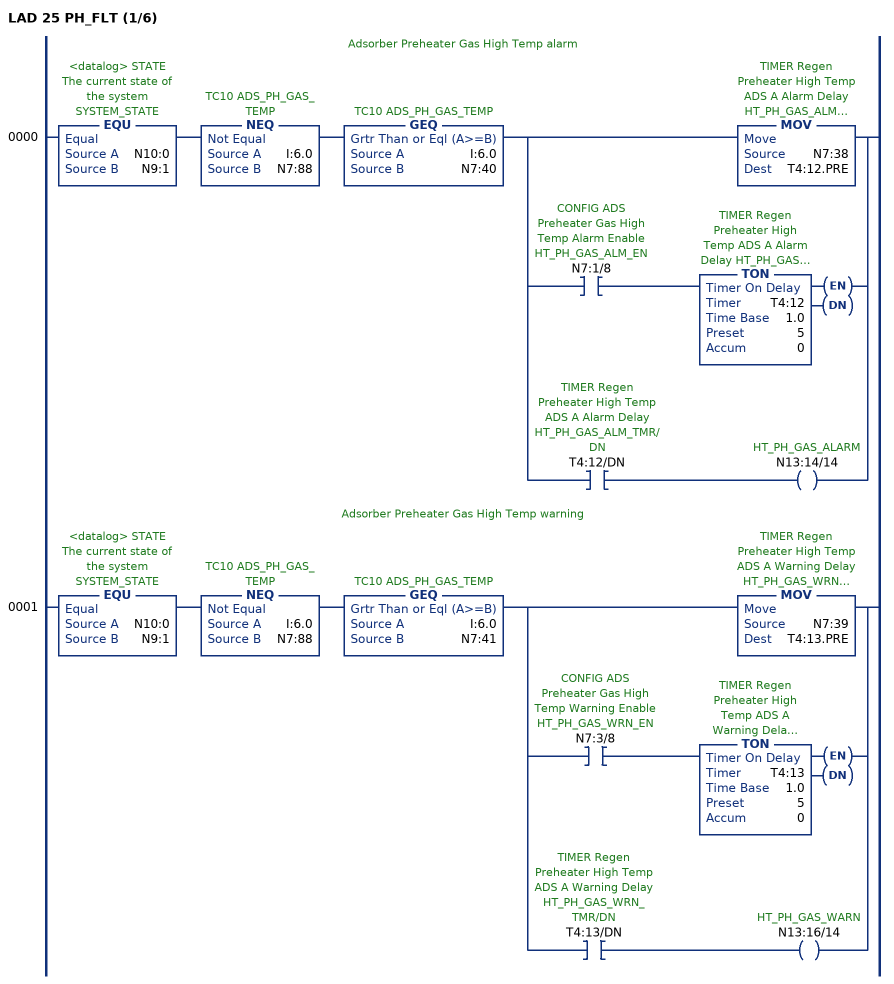
% Rung: 0 %
% Adsorber Preheater Gas High Temp alarm %
SOR EQU N10:0 N9:1 NEQ I:6.0 N7:88 GEQ I:6.0 N7:40 BST MOV N7:38 T4:12.PRE NXB XIC N7:1/8 TON T4:12 1.0 5 0 NXB XIC T4:12/DN OTE N13:14/14 BND EOR
%   N10:0  SYSTEM_STATE  "<datalog> STATE The current state of the system" %
%   N9:1  SYSTEM_PROCESS  "STATE System Process" %
%   I:6.0  ADS_PH_GAS_TEMP  "TC10" %
%   N7:88  TC_OPEN_SP  "CONFIG TC Open Setpoint" %
%   N7:40  HT_PH_GAS_ALM_SP  "CONFIG ADS Preheater Gas High Temp Alarm Setpoint" %
%   N7:38  HT_PH_GAS_ALM_DLY  "CONFIG ADS Preheater Gas High Temp Alarm Delay" %
%   T4:12  HT_PH_GAS_ALM_TMR  "TIMER Regen Preheater High Temp ADS A Alarm Delay" %
%   N7:1/8  HT_PH_GAS_ALM_EN  "CONFIG ADS Preheater Gas High Temp Alarm Enable" %
%   N13:14/14  HT_PH_GAS_ALARM %
% Rung: 1 %
% Adsorber Preheater Gas High Temp warning %
SOR EQU N10:0 N9:1 NEQ I:6.0 N7:88 GEQ I:6.0 N7:41 BST MOV N7:39 T4:13.PRE NXB XIC N7:3/8 TON T4:13 1.0 5 0 NXB XIC T4:13/DN OTE N13:16/14 BND EOR
%   N10:0  SYSTEM_STATE  "<datalog> STATE The current state of the system" %
%   N9:1  SYSTEM_PROCESS  "STATE System Process" %
%   I:6.0  ADS_PH_GAS_TEMP  "TC10" %
%   N7:88  TC_OPEN_SP  "CONFIG TC Open Setpoint" %
%   N7:41  HT_PH_GAS_WRN_SP  "CONFIG ADS Preheater Gas High Temp Warning Setpoint" %
%   N7:39  HT_PH_GAS_WRN_DLY  "CONFIG ADS Preheater Gas High Temp Warning Delay" %
%   T4:13  HT_PH_GAS_WRN_TMR  "TIMER Regen Preheater High Temp ADS A Warning Delay" %
%   N7:3/8  HT_PH_GAS_WRN_EN  "CONFIG ADS Preheater Gas High Temp Warning Enable" %
%   N13:16/14  HT_PH_GAS_WARN %

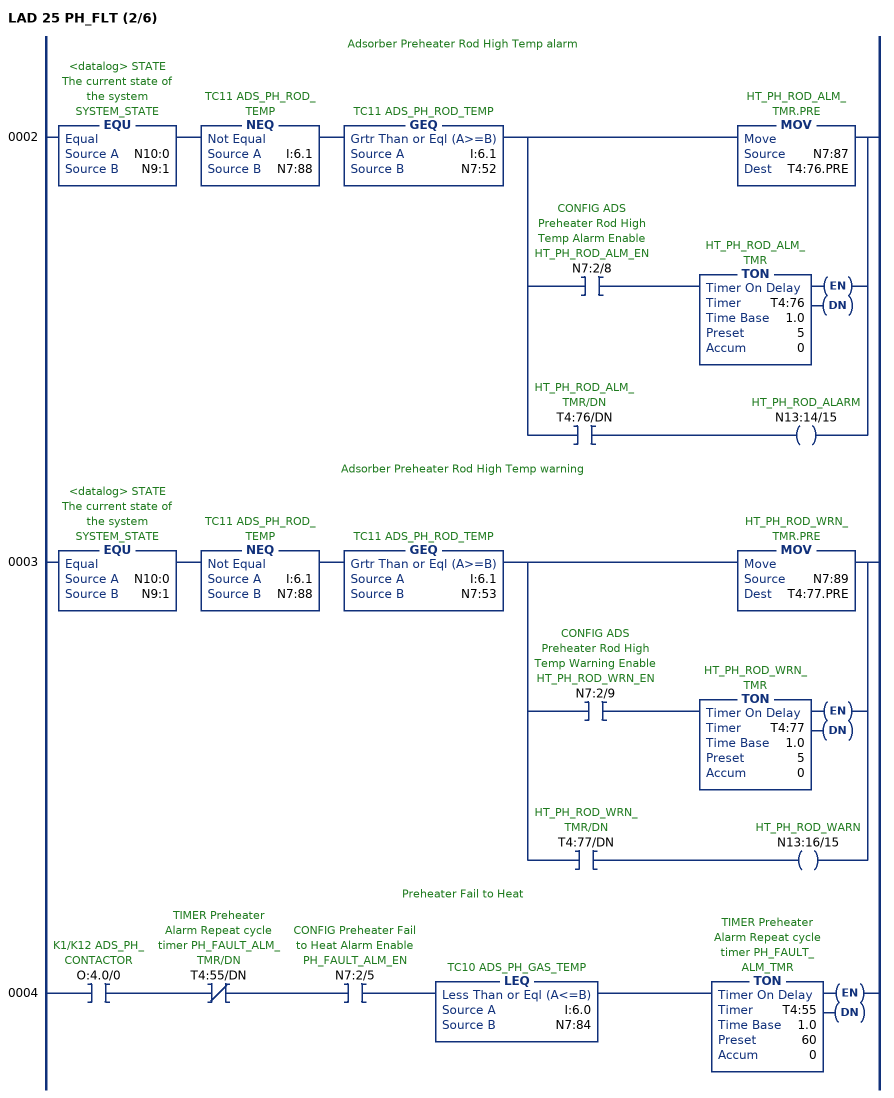
% Rung: 2 %
% Adsorber Preheater Rod High Temp alarm %
SOR EQU N10:0 N9:1 NEQ I:6.1 N7:88 GEQ I:6.1 N7:52 BST MOV N7:87 T4:76.PRE NXB XIC N7:2/8 TON T4:76 1.0 5 0 NXB XIC T4:76/DN OTE N13:14/15 BND EOR
%   N10:0  SYSTEM_STATE  "<datalog> STATE The current state of the system" %
%   N9:1  SYSTEM_PROCESS  "STATE System Process" %
%   I:6.1  ADS_PH_ROD_TEMP  "TC11" %
%   N7:88  TC_OPEN_SP  "CONFIG TC Open Setpoint" %
%   N7:52  HT_PH_ROD_ALM_SP  "CONFIG ADS Preheater Rod High Temp Alarm Setpoint" %
%   N7:87  HT_PH_ROD_ALM_DLY  "CONFIG ADS Preheater Rod High Temp Alarm Delay" %
%   T4:76  HT_PH_ROD_ALM_TMR %
%   N7:2/8  HT_PH_ROD_ALM_EN  "CONFIG ADS Preheater Rod High Temp Alarm Enable" %
%   N13:14/15  HT_PH_ROD_ALARM %
% Rung: 3 %
% Adsorber Preheater Rod High Temp warning %
SOR EQU N10:0 N9:1 NEQ I:6.1 N7:88 GEQ I:6.1 N7:53 BST MOV N7:89 T4:77.PRE NXB XIC N7:2/9 TON T4:77 1.0 5 0 NXB XIC T4:77/DN OTE N13:16/15 BND EOR
%   N10:0  SYSTEM_STATE  "<datalog> STATE The current state of the system" %
%   N9:1  SYSTEM_PROCESS  "STATE System Process" %
%   I:6.1  ADS_PH_ROD_TEMP  "TC11" %
%   N7:88  TC_OPEN_SP  "CONFIG TC Open Setpoint" %
%   N7:53  HT_PH_ROD_WRN_SP  "CONFIG ADS Preheater Rod High Temp Warning Setpoint" %
%   N7:89  HT_PH_ROD_WRN_DLY  "CONFIG ADS Preheater Rod High Temp Warning Delay" %
%   T4:77  HT_PH_ROD_WRN_TMR %
%   N7:2/9  HT_PH_ROD_WRN_EN  "CONFIG ADS Preheater Rod High Temp Warning Enable" %
%   N13:16/15  HT_PH_ROD_WARN %
% Rung: 4 %
% Preheater Fail to Heat %
SOR XIC O:4.0/0 XIO T4:55/DN XIC N7:2/5 LEQ I:6.0 N7:84 TON T4:55 1.0 60 0 EOR
%   O:4.0/0  ADS_PH_CONTACTOR  "K1/K12" %
%   T4:55  PH_FAULT_ALM_TMR  "TIMER Preheater Alarm Repeat cycle timer" %
%   N7:2/5  PH_FAULT_ALM_EN  "CONFIG Preheater Fail to Heat Alarm Enable" %
%   I:6.0  ADS_PH_GAS_TEMP  "TC10" %
%   N7:84  PH_FAULT_ALARM_SP  "CONFIG Preheater Fail to Heat Alarm Setpoint" %

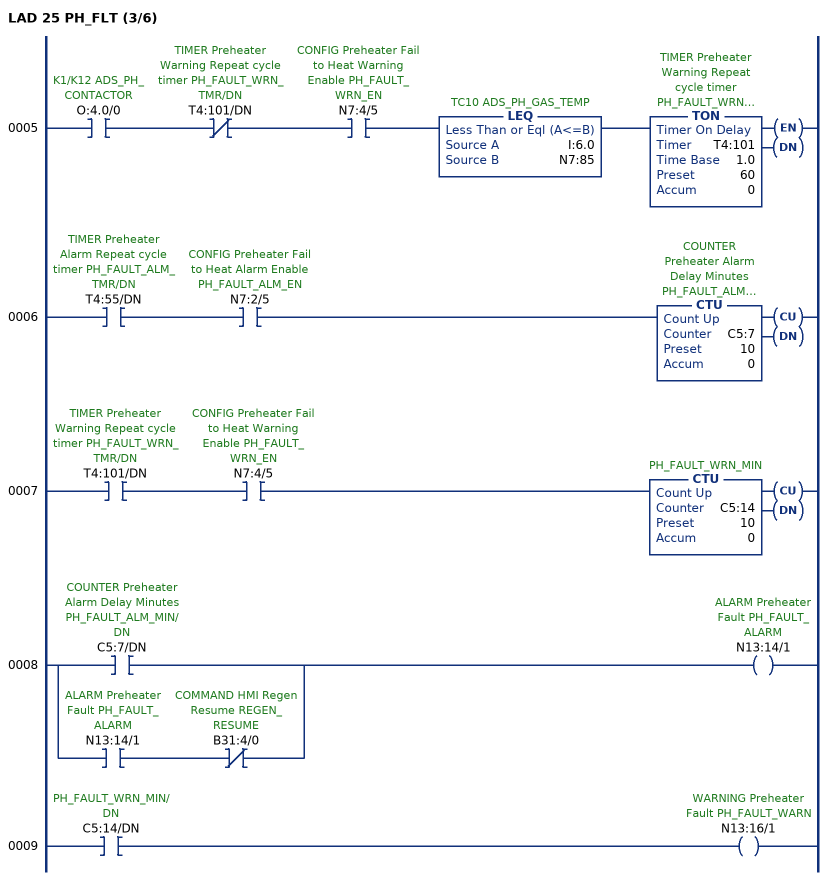
% Rung: 5 %
SOR XIC O:4.0/0 XIO T4:101/DN XIC N7:4/5 LEQ I:6.0 N7:85 TON T4:101 1.0 60 0 EOR
%   O:4.0/0  ADS_PH_CONTACTOR  "K1/K12" %
%   T4:101  PH_FAULT_WRN_TMR  "TIMER Preheater Warning Repeat cycle timer" %
%   N7:4/5  PH_FAULT_WRN_EN  "CONFIG Preheater Fail to Heat Warning Enable" %
%   I:6.0  ADS_PH_GAS_TEMP  "TC10" %
%   N7:85  PH_FAULT_WARN_SP  "CONFIG Preheater Fail to Heat Warning Setpoint" %
% Rung: 6 %
SOR XIC T4:55/DN XIC N7:2/5 CTU C5:7 10 0 EOR
%   T4:55  PH_FAULT_ALM_TMR  "TIMER Preheater Alarm Repeat cycle timer" %
%   N7:2/5  PH_FAULT_ALM_EN  "CONFIG Preheater Fail to Heat Alarm Enable" %
%   C5:7  PH_FAULT_ALM_MIN  "COUNTER Preheater Alarm Delay Minutes" %
% Rung: 7 %
SOR XIC T4:101/DN XIC N7:4/5 CTU C5:14 10 0 EOR
%   T4:101  PH_FAULT_WRN_TMR  "TIMER Preheater Warning Repeat cycle timer" %
%   N7:4/5  PH_FAULT_WRN_EN  "CONFIG Preheater Fail to Heat Warning Enable" %
%   C5:14  PH_FAULT_WRN_MIN %
% Rung: 8 %
SOR BST XIC C5:7/DN NXB XIC N13:14/1 XIO B31:4/0 BND OTE N13:14/1 EOR
%   C5:7  PH_FAULT_ALM_MIN  "COUNTER Preheater Alarm Delay Minutes" %
%   N13:14/1  PH_FAULT_ALARM  "ALARM Preheater Fault" %
%   B31:4/0  REGEN_RESUME  "COMMAND HMI Regen Resume" %
% Rung: 9 %
SOR XIC C5:14/DN OTE N13:16/1 EOR
%   C5:14  PH_FAULT_WRN_MIN %
%   N13:16/1  PH_FAULT_WARN  "WARNING Preheater Fault" %

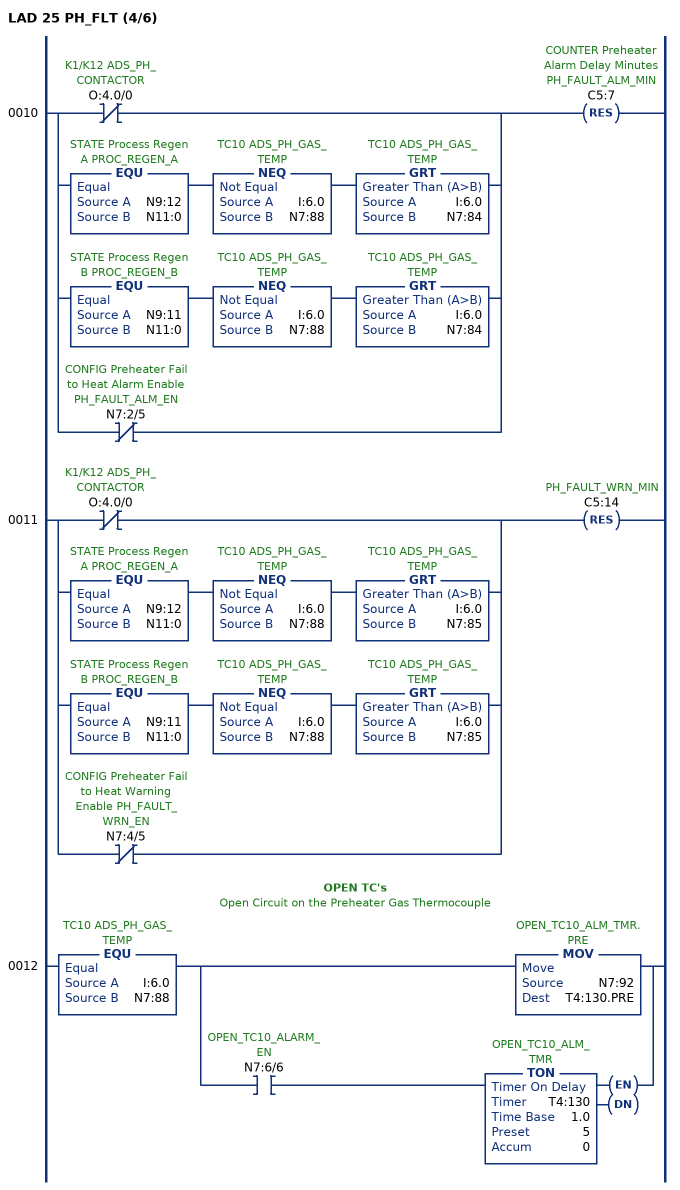
% Rung: 10 %
SOR BST XIO O:4.0/0 NXB EQU N9:12 N11:0 NEQ I:6.0 N7:88 GRT I:6.0 N7:84 NXB EQU N9:11 N11:0 NEQ I:6.0 N7:88 GRT I:6.0 N7:84 NXB XIO N7:2/5 BND RES C5:7 EOR
%   O:4.0/0  ADS_PH_CONTACTOR  "K1/K12" %
%   N9:12  PROC_REGEN_A  "STATE Process Regen A" %
%   N11:0  PROC_STATE  "<datalog> STATE The current state of the process" %
%   I:6.0  ADS_PH_GAS_TEMP  "TC10" %
%   N7:88  TC_OPEN_SP  "CONFIG TC Open Setpoint" %
%   N7:84  PH_FAULT_ALARM_SP  "CONFIG Preheater Fail to Heat Alarm Setpoint" %
%   N9:11  PROC_REGEN_B  "STATE Process Regen B" %
%   N7:2/5  PH_FAULT_ALM_EN  "CONFIG Preheater Fail to Heat Alarm Enable" %
%   C5:7  PH_FAULT_ALM_MIN  "COUNTER Preheater Alarm Delay Minutes" %
% Rung: 11 %
SOR BST XIO O:4.0/0 NXB EQU N9:12 N11:0 NEQ I:6.0 N7:88 GRT I:6.0 N7:85 NXB EQU N9:11 N11:0 NEQ I:6.0 N7:88 GRT I:6.0 N7:85 NXB XIO N7:4/5 BND RES C5:14 EOR
%   O:4.0/0  ADS_PH_CONTACTOR  "K1/K12" %
%   N9:12  PROC_REGEN_A  "STATE Process Regen A" %
%   N11:0  PROC_STATE  "<datalog> STATE The current state of the process" %
%   I:6.0  ADS_PH_GAS_TEMP  "TC10" %
%   N7:88  TC_OPEN_SP  "CONFIG TC Open Setpoint" %
%   N7:85  PH_FAULT_WARN_SP  "CONFIG Preheater Fail to Heat Warning Setpoint" %
%   N9:11  PROC_REGEN_B  "STATE Process Regen B" %
%   N7:4/5  PH_FAULT_WRN_EN  "CONFIG Preheater Fail to Heat Warning Enable" %
%   C5:14  PH_FAULT_WRN_MIN %
% Rung: 12 %
% TITLE: OPEN TC's %
% Open Circuit on the Preheater Gas Thermocouple %
SOR EQU I:6.0 N7:88 BST MOV N7:92 T4:130.PRE NXB XIC N7:6/6 TON T4:130 1.0 5 0 BND EOR
%   I:6.0  ADS_PH_GAS_TEMP  "TC10" %
%   N7:88  TC_OPEN_SP  "CONFIG TC Open Setpoint" %
%   N7:92  OPEN_TC_ALM_DLY  "CONFIG TC Open Alarm Delay" %
%   T4:130  OPEN_TC10_ALM_TMR %
%   N7:6/6  OPEN_TC10_ALARM_EN %

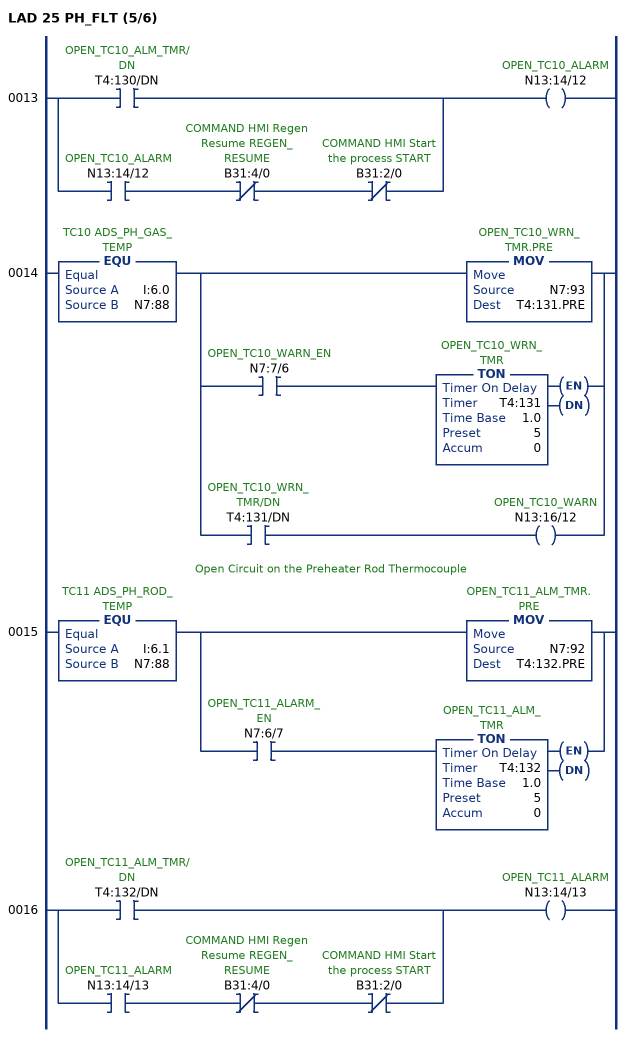
% Rung: 13 %
SOR BST XIC T4:130/DN NXB XIC N13:14/12 XIO B31:4/0 XIO B31:2/0 BND OTE N13:14/12 EOR
%   T4:130  OPEN_TC10_ALM_TMR %
%   N13:14/12  OPEN_TC10_ALARM %
%   B31:4/0  REGEN_RESUME  "COMMAND HMI Regen Resume" %
%   B31:2/0  START  "COMMAND HMI Start the process" %
% Rung: 14 %
SOR EQU I:6.0 N7:88 BST MOV N7:93 T4:131.PRE NXB XIC N7:7/6 TON T4:131 1.0 5 0 NXB XIC T4:131/DN OTE N13:16/12 BND EOR
%   I:6.0  ADS_PH_GAS_TEMP  "TC10" %
%   N7:88  TC_OPEN_SP  "CONFIG TC Open Setpoint" %
%   N7:93  OPEN_TC_WRN_DLY  "CONFIG TC Open Warning Delay" %
%   T4:131  OPEN_TC10_WRN_TMR %
%   N7:7/6  OPEN_TC10_WARN_EN %
%   N13:16/12  OPEN_TC10_WARN %
% Rung: 15 %
% Open Circuit on the Preheater Rod Thermocouple %
SOR EQU I:6.1 N7:88 BST MOV N7:92 T4:132.PRE NXB XIC N7:6/7 TON T4:132 1.0 5 0 BND EOR
%   I:6.1  ADS_PH_ROD_TEMP  "TC11" %
%   N7:88  TC_OPEN_SP  "CONFIG TC Open Setpoint" %
%   N7:92  OPEN_TC_ALM_DLY  "CONFIG TC Open Alarm Delay" %
%   T4:132  OPEN_TC11_ALM_TMR %
%   N7:6/7  OPEN_TC11_ALARM_EN %
% Rung: 16 %
SOR BST XIC T4:132/DN NXB XIC N13:14/13 XIO B31:4/0 XIO B31:2/0 BND OTE N13:14/13 EOR
%   T4:132  OPEN_TC11_ALM_TMR %
%   N13:14/13  OPEN_TC11_ALARM %
%   B31:4/0  REGEN_RESUME  "COMMAND HMI Regen Resume" %
%   B31:2/0  START  "COMMAND HMI Start the process" %

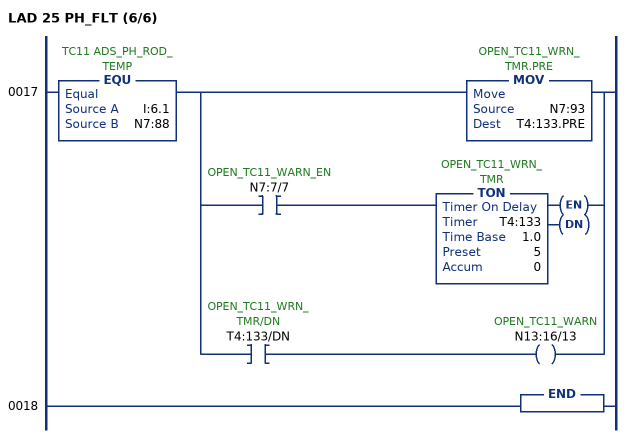
% Rung: 17 %
SOR EQU I:6.1 N7:88 BST MOV N7:93 T4:133.PRE NXB XIC N7:7/7 TON T4:133 1.0 5 0 NXB XIC T4:133/DN OTE N13:16/13 BND EOR
%   I:6.1  ADS_PH_ROD_TEMP  "TC11" %
%   N7:88  TC_OPEN_SP  "CONFIG TC Open Setpoint" %
%   N7:93  OPEN_TC_WRN_DLY  "CONFIG TC Open Warning Delay" %
%   T4:133  OPEN_TC11_WRN_TMR %
%   N7:7/7  OPEN_TC11_WARN_EN %
%   N13:16/13  OPEN_TC11_WARN %
% Rung: 18 %
SOR END EOR

LADDER 26 "ADS_C"
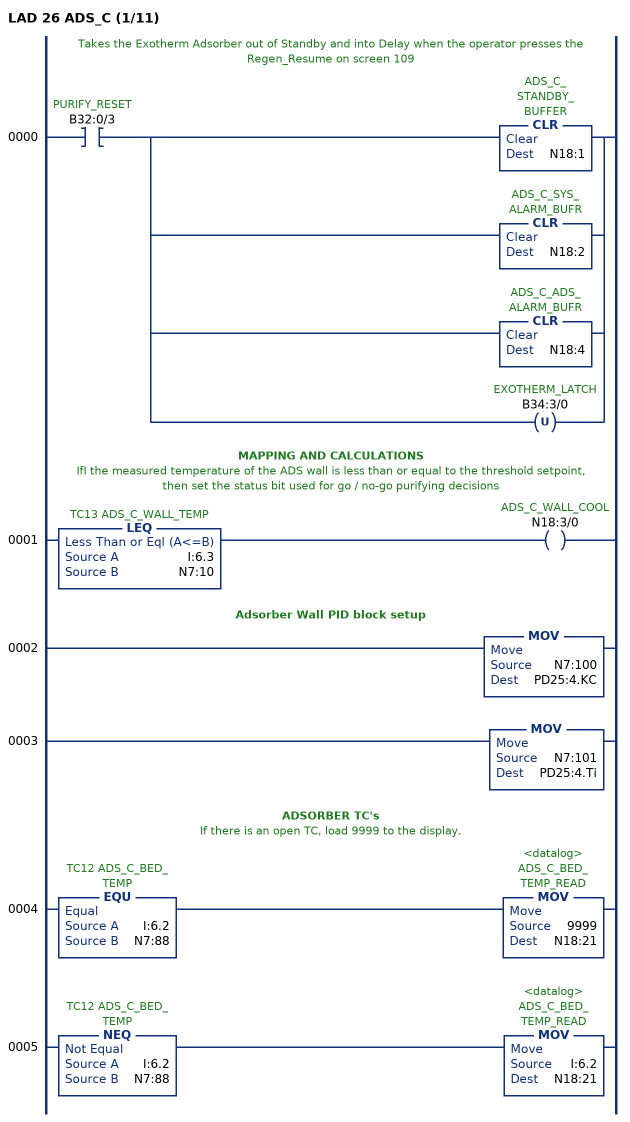
% Rung: 0 %
% Takes the Exotherm Adsorber out of Standby and into Delay when the operator presses the Regen_Resume on screen 109 %
SOR XIC B32:0/3 BST CLR N18:1 NXB CLR N18:2 NXB CLR N18:4 NXB OTU B34:3/0 BND EOR
%   B32:0/3  PURIFY_RESET %
%   N18:1  ADS_C_STANDBY_BUFFER %
%   N18:2  ADS_C_SYS_ALARM_BUFR %
%   N18:4  ADS_C_ADS_ALARM_BUFR %
%   B34:3/0  EXOTHERM_LATCH %
% Rung: 1 %
% TITLE: MAPPING AND CALCULATIONS %
% IfI the measured temperature of the ADS wall is less than or equal to the threshold setpoint, then set the status bit used for go / no-go purifying decisions %
SOR LEQ I:6.3 N7:10 OTE N18:3/0 EOR
%   I:6.3  ADS_C_WALL_TEMP  "TC13" %
%   N7:10  ADS_WALL_TEMP_COOL  "CONFIG The temp at which the adsorber wall is deemed to be cool enough to purify" %
%   N18:3/0  ADS_C_WALL_COOL %
% Rung: 2 %
% TITLE: Adsorber Wall PID block setup %
SOR MOV N7:100 PD25:4.KC EOR
%   N7:100  BLANKET_P  "CONFIG Blanket Proportional Gain" %
% Rung: 3 %
SOR MOV N7:101 PD25:4.Ti EOR
%   N7:101  BLANKET_I  "CONFIG Blanket Integral Gain" %
% Rung: 4 %
% TITLE: ADSORBER TC's %
% If there is an open TC, load 9999 to the display. %
SOR EQU I:6.2 N7:88 MOV 9999 N18:21 EOR
%   I:6.2  ADS_C_BED_TEMP  "TC12" %
%   N7:88  TC_OPEN_SP  "CONFIG TC Open Setpoint" %
%   N18:21  ADS_C_BED_TEMP_READ  "<datalog>" %
% Rung: 5 %
SOR NEQ I:6.2 N7:88 MOV I:6.2 N18:21 EOR
%   I:6.2  ADS_C_BED_TEMP  "TC12" %
%   N7:88  TC_OPEN_SP  "CONFIG TC Open Setpoint" %
%   N18:21  ADS_C_BED_TEMP_READ  "<datalog>" %

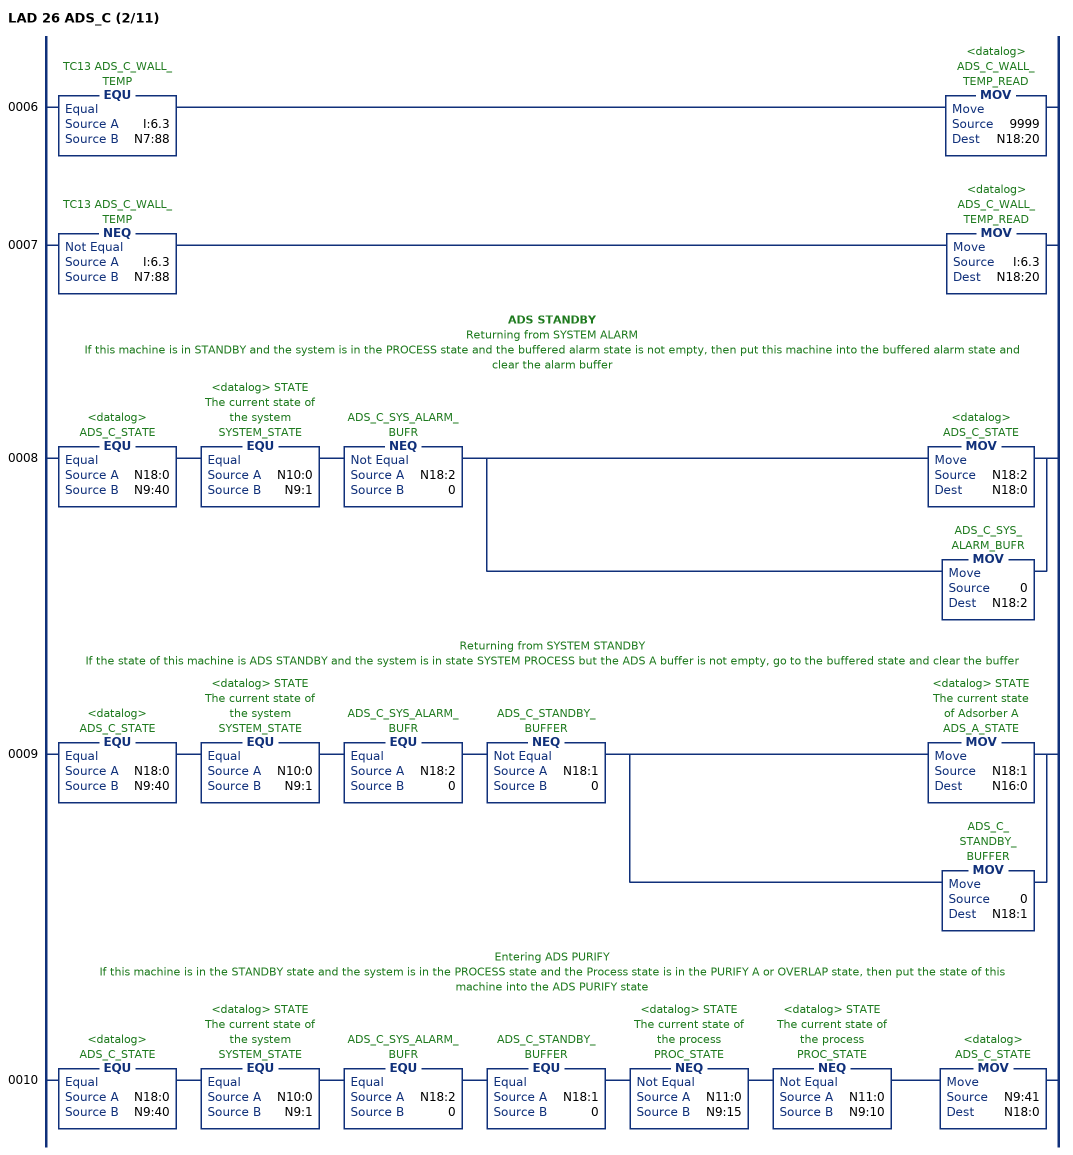
% Rung: 6 %
SOR EQU I:6.3 N7:88 MOV 9999 N18:20 EOR
%   I:6.3  ADS_C_WALL_TEMP  "TC13" %
%   N7:88  TC_OPEN_SP  "CONFIG TC Open Setpoint" %
%   N18:20  ADS_C_WALL_TEMP_READ  "<datalog>" %
% Rung: 7 %
SOR NEQ I:6.3 N7:88 MOV I:6.3 N18:20 EOR
%   I:6.3  ADS_C_WALL_TEMP  "TC13" %
%   N7:88  TC_OPEN_SP  "CONFIG TC Open Setpoint" %
%   N18:20  ADS_C_WALL_TEMP_READ  "<datalog>" %
% Rung: 8 %
% TITLE: ADS STANDBY %
% Returning from SYSTEM ALARM
% If this machine is in STANDBY and the system is in the PROCESS state and the buffered alarm state is not empty, then put this machine into the buffered alarm state and clear the alarm buffer %
SOR EQU N18:0 N9:40 EQU N10:0 N9:1 NEQ N18:2 0 BST MOV N18:2 N18:0 NXB MOV 0 N18:2 BND EOR
%   N18:0  ADS_C_STATE  "<datalog>" %
%   N9:40  ADS_STANDBY  "STATE ADS Standby" %
%   N10:0  SYSTEM_STATE  "<datalog> STATE The current state of the system" %
%   N9:1  SYSTEM_PROCESS  "STATE System Process" %
%   N18:2  ADS_C_SYS_ALARM_BUFR %
% Rung: 9 %
% Returning from SYSTEM STANDBY
% If the state of this machine is ADS STANDBY and the system is in state SYSTEM PROCESS but the ADS A buffer is not empty, go to the buffered state and clear the buffer %
SOR EQU N18:0 N9:40 EQU N10:0 N9:1 EQU N18:2 0 NEQ N18:1 0 BST MOV N18:1 N16:0 NXB MOV 0 N18:1 BND EOR
%   N18:0  ADS_C_STATE  "<datalog>" %
%   N9:40  ADS_STANDBY  "STATE ADS Standby" %
%   N10:0  SYSTEM_STATE  "<datalog> STATE The current state of the system" %
%   N9:1  SYSTEM_PROCESS  "STATE System Process" %
%   N18:2  ADS_C_SYS_ALARM_BUFR %
%   N18:1  ADS_C_STANDBY_BUFFER %
%   N16:0  ADS_A_STATE  "<datalog> STATE The current state of Adsorber A" %
% Rung: 10 %
% Entering ADS PURIFY
% If this machine is in the STANDBY state and the system is in the PROCESS state and the Process state is in the PURIFY A or OVERLAP state, then put the state of this machine into the ADS PURIFY state %
SOR EQU N18:0 N9:40 EQU N10:0 N9:1 EQU N18:2 0 EQU N18:1 0 NEQ N11:0 N9:15 NEQ N11:0 N9:10 MOV N9:41 N18:0 EOR
%   N18:0  ADS_C_STATE  "<datalog>" %
%   N9:40  ADS_STANDBY  "STATE ADS Standby" %
%   N10:0  SYSTEM_STATE  "<datalog> STATE The current state of the system" %
%   N9:1  SYSTEM_PROCESS  "STATE System Process" %
%   N18:2  ADS_C_SYS_ALARM_BUFR %
%   N18:1  ADS_C_STANDBY_BUFFER %
%   N11:0  PROC_STATE  "<datalog> STATE The current state of the process" %
%   N9:15  PROC_REGEN_C  "STATE Process Regen C" %
%   N9:10  PROCESS_STANDBY  "STATE Process Standby" %
%   N9:41  ADS_PURIFY  "STATE ADS Purify" %

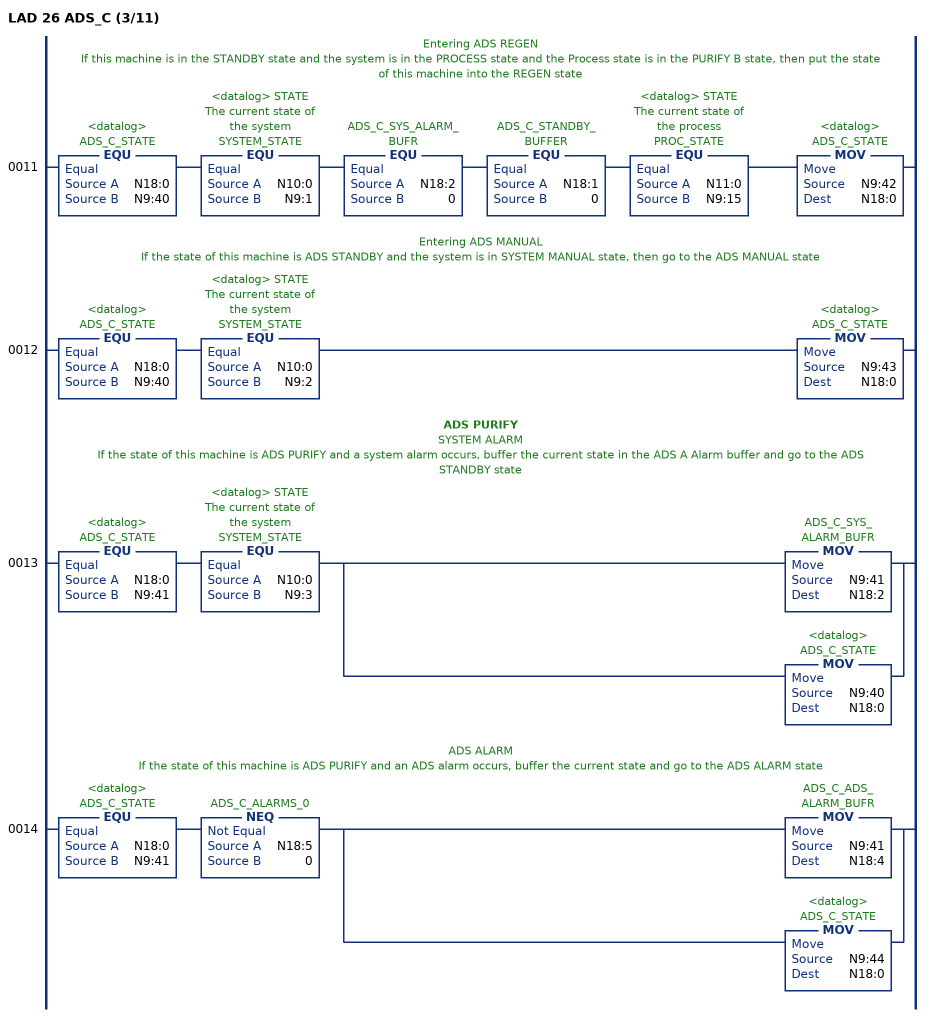
% Rung: 11 %
% Entering ADS REGEN
% If this machine is in the STANDBY state and the system is in the PROCESS state and the Process state is in the PURIFY B state, then put the state of this machine into the REGEN state %
SOR EQU N18:0 N9:40 EQU N10:0 N9:1 EQU N18:2 0 EQU N18:1 0 EQU N11:0 N9:15 MOV N9:42 N18:0 EOR
%   N18:0  ADS_C_STATE  "<datalog>" %
%   N9:40  ADS_STANDBY  "STATE ADS Standby" %
%   N10:0  SYSTEM_STATE  "<datalog> STATE The current state of the system" %
%   N9:1  SYSTEM_PROCESS  "STATE System Process" %
%   N18:2  ADS_C_SYS_ALARM_BUFR %
%   N18:1  ADS_C_STANDBY_BUFFER %
%   N11:0  PROC_STATE  "<datalog> STATE The current state of the process" %
%   N9:15  PROC_REGEN_C  "STATE Process Regen C" %
%   N9:42  ADS_REGEN  "STATE ADS Regen" %
% Rung: 12 %
% Entering ADS MANUAL
% If the state of this machine is ADS STANDBY and the system is in SYSTEM MANUAL state, then go to the ADS MANUAL state %
SOR EQU N18:0 N9:40 EQU N10:0 N9:2 MOV N9:43 N18:0 EOR
%   N18:0  ADS_C_STATE  "<datalog>" %
%   N9:40  ADS_STANDBY  "STATE ADS Standby" %
%   N10:0  SYSTEM_STATE  "<datalog> STATE The current state of the system" %
%   N9:2  SYSTEM_MANUAL  "STATE System Manual" %
%   N9:43  ADS_MANUAL  "STATE ADS Manual" %
% Rung: 13 %
% TITLE: ADS PURIFY %
% SYSTEM ALARM
% If the state of this machine is ADS PURIFY and a system alarm occurs, buffer the current state in the ADS A Alarm buffer and go to the ADS STANDBY state %
SOR EQU N18:0 N9:41 EQU N10:0 N9:3 BST MOV N9:41 N18:2 NXB MOV N9:40 N18:0 BND EOR
%   N18:0  ADS_C_STATE  "<datalog>" %
%   N9:41  ADS_PURIFY  "STATE ADS Purify" %
%   N10:0  SYSTEM_STATE  "<datalog> STATE The current state of the system" %
%   N9:3  SYSTEM_ALARM  "STATE System Alarm" %
%   N18:2  ADS_C_SYS_ALARM_BUFR %
%   N9:40  ADS_STANDBY  "STATE ADS Standby" %
% Rung: 14 %
% ADS ALARM
% If the state of this machine is ADS PURIFY and an ADS alarm occurs, buffer the current state and go to the ADS ALARM state %
SOR EQU N18:0 N9:41 NEQ N18:5 0 BST MOV N9:41 N18:4 NXB MOV N9:44 N18:0 BND EOR
%   N18:0  ADS_C_STATE  "<datalog>" %
%   N9:41  ADS_PURIFY  "STATE ADS Purify" %
%   N18:5  ADS_C_ALARMS_0 %
%   N18:4  ADS_C_ADS_ALARM_BUFR %
%   N9:44  ADS_ALARM  "STATE ADS Alarm" %

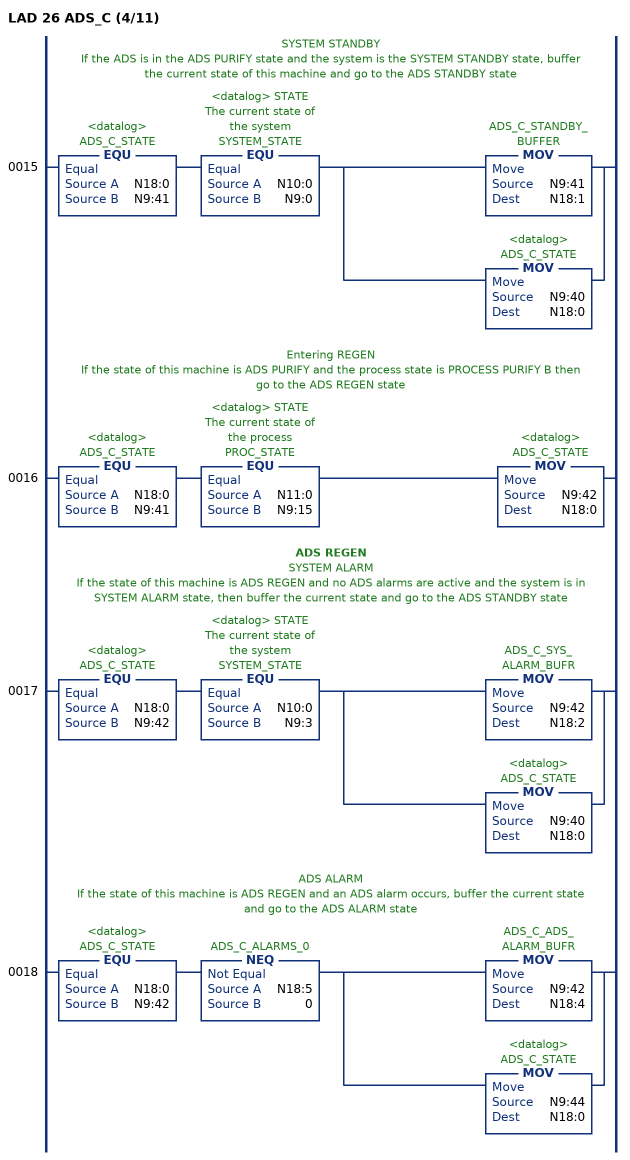
% Rung: 15 %
% SYSTEM STANDBY
% If the ADS is in the ADS PURIFY state and the system is the SYSTEM STANDBY state, buffer the current state of this machine and go to the ADS STANDBY state %
SOR EQU N18:0 N9:41 EQU N10:0 N9:0 BST MOV N9:41 N18:1 NXB MOV N9:40 N18:0 BND EOR
%   N18:0  ADS_C_STATE  "<datalog>" %
%   N9:41  ADS_PURIFY  "STATE ADS Purify" %
%   N10:0  SYSTEM_STATE  "<datalog> STATE The current state of the system" %
%   N9:0  SYSTEM_STANDBY  "STATE System Standby" %
%   N18:1  ADS_C_STANDBY_BUFFER %
%   N9:40  ADS_STANDBY  "STATE ADS Standby" %
% Rung: 16 %
% Entering REGEN
% If the state of this machine is ADS PURIFY and the process state is PROCESS PURIFY B then go to the ADS REGEN state %
SOR EQU N18:0 N9:41 EQU N11:0 N9:15 MOV N9:42 N18:0 EOR
%   N18:0  ADS_C_STATE  "<datalog>" %
%   N9:41  ADS_PURIFY  "STATE ADS Purify" %
%   N11:0  PROC_STATE  "<datalog> STATE The current state of the process" %
%   N9:15  PROC_REGEN_C  "STATE Process Regen C" %
%   N9:42  ADS_REGEN  "STATE ADS Regen" %
% Rung: 17 %
% TITLE: ADS REGEN %
% SYSTEM ALARM
% If the state of this machine is ADS REGEN and no ADS alarms are active and the system is in SYSTEM ALARM state, then buffer the current state and go to the ADS STANDBY state %
SOR EQU N18:0 N9:42 EQU N10:0 N9:3 BST MOV N9:42 N18:2 NXB MOV N9:40 N18:0 BND EOR
%   N18:0  ADS_C_STATE  "<datalog>" %
%   N9:42  ADS_REGEN  "STATE ADS Regen" %
%   N10:0  SYSTEM_STATE  "<datalog> STATE The current state of the system" %
%   N9:3  SYSTEM_ALARM  "STATE System Alarm" %
%   N18:2  ADS_C_SYS_ALARM_BUFR %
%   N9:40  ADS_STANDBY  "STATE ADS Standby" %
% Rung: 18 %
% ADS ALARM
% If the state of this machine is ADS REGEN and an ADS alarm occurs, buffer the current state and go to the ADS ALARM state %
SOR EQU N18:0 N9:42 NEQ N18:5 0 BST MOV N9:42 N18:4 NXB MOV N9:44 N18:0 BND EOR
%   N18:0  ADS_C_STATE  "<datalog>" %
%   N9:42  ADS_REGEN  "STATE ADS Regen" %
%   N18:5  ADS_C_ALARMS_0 %
%   N18:4  ADS_C_ADS_ALARM_BUFR %
%   N9:44  ADS_ALARM  "STATE ADS Alarm" %

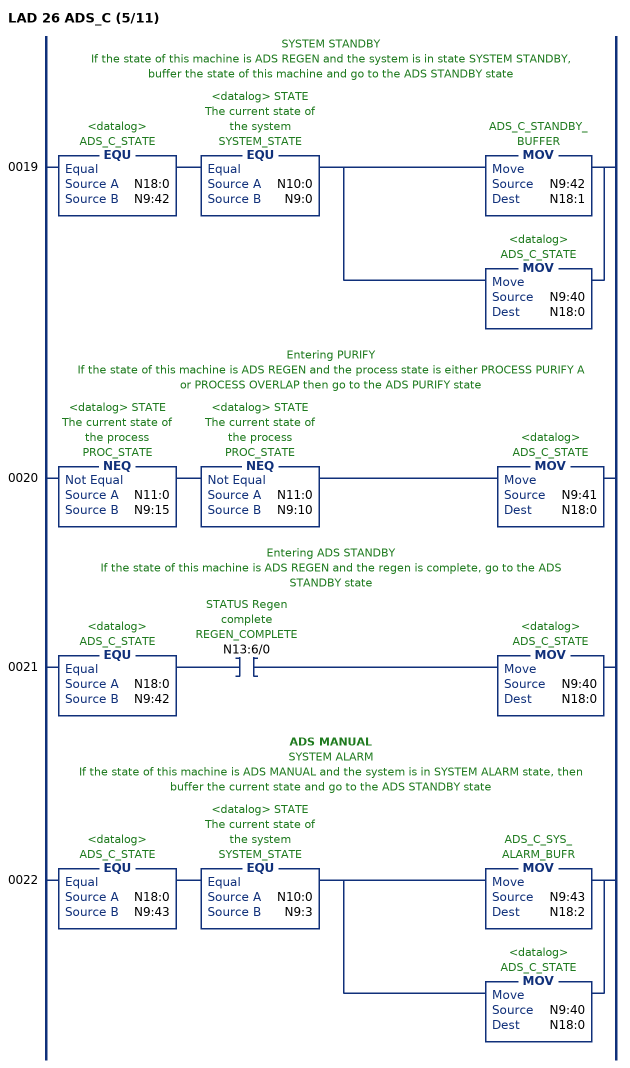
% Rung: 19 %
% SYSTEM STANDBY
% If the state of this machine is ADS REGEN and the system is in state SYSTEM STANDBY, buffer the state of this machine and go to the ADS STANDBY state %
SOR EQU N18:0 N9:42 EQU N10:0 N9:0 BST MOV N9:42 N18:1 NXB MOV N9:40 N18:0 BND EOR
%   N18:0  ADS_C_STATE  "<datalog>" %
%   N9:42  ADS_REGEN  "STATE ADS Regen" %
%   N10:0  SYSTEM_STATE  "<datalog> STATE The current state of the system" %
%   N9:0  SYSTEM_STANDBY  "STATE System Standby" %
%   N18:1  ADS_C_STANDBY_BUFFER %
%   N9:40  ADS_STANDBY  "STATE ADS Standby" %
% Rung: 20 %
% Entering PURIFY
% If the state of this machine is ADS REGEN and the process state is either PROCESS PURIFY A or PROCESS OVERLAP then go to the ADS PURIFY state %
SOR NEQ N11:0 N9:15 NEQ N11:0 N9:10 MOV N9:41 N18:0 EOR
%   N11:0  PROC_STATE  "<datalog> STATE The current state of the process" %
%   N9:15  PROC_REGEN_C  "STATE Process Regen C" %
%   N9:10  PROCESS_STANDBY  "STATE Process Standby" %
%   N9:41  ADS_PURIFY  "STATE ADS Purify" %
%   N18:0  ADS_C_STATE  "<datalog>" %
% Rung: 21 %
% Entering ADS STANDBY
% If the state of this machine is ADS REGEN and the regen is complete, go to the ADS STANDBY state %
SOR EQU N18:0 N9:42 XIC N13:6/0 MOV N9:40 N18:0 EOR
%   N18:0  ADS_C_STATE  "<datalog>" %
%   N9:42  ADS_REGEN  "STATE ADS Regen" %
%   N13:6/0  REGEN_COMPLETE  "STATUS Regen complete" %
%   N9:40  ADS_STANDBY  "STATE ADS Standby" %
% Rung: 22 %
% TITLE: ADS MANUAL %
% SYSTEM ALARM
% If the state of this machine is ADS MANUAL and the system is in SYSTEM ALARM state, then buffer the current state and go to the ADS STANDBY state %
SOR EQU N18:0 N9:43 EQU N10:0 N9:3 BST MOV N9:43 N18:2 NXB MOV N9:40 N18:0 BND EOR
%   N18:0  ADS_C_STATE  "<datalog>" %
%   N9:43  ADS_MANUAL  "STATE ADS Manual" %
%   N10:0  SYSTEM_STATE  "<datalog> STATE The current state of the system" %
%   N9:3  SYSTEM_ALARM  "STATE System Alarm" %
%   N18:2  ADS_C_SYS_ALARM_BUFR %
%   N9:40  ADS_STANDBY  "STATE ADS Standby" %

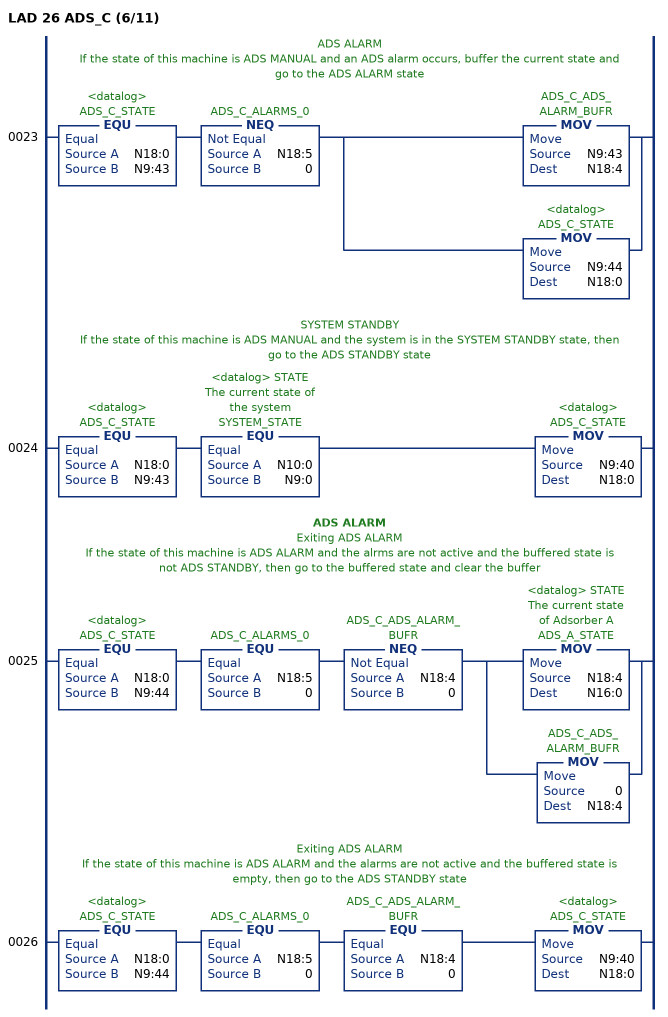
% Rung: 23 %
% ADS ALARM
% If the state of this machine is ADS MANUAL and an ADS alarm occurs, buffer the current state and go to the ADS ALARM state %
SOR EQU N18:0 N9:43 NEQ N18:5 0 BST MOV N9:43 N18:4 NXB MOV N9:44 N18:0 BND EOR
%   N18:0  ADS_C_STATE  "<datalog>" %
%   N9:43  ADS_MANUAL  "STATE ADS Manual" %
%   N18:5  ADS_C_ALARMS_0 %
%   N18:4  ADS_C_ADS_ALARM_BUFR %
%   N9:44  ADS_ALARM  "STATE ADS Alarm" %
% Rung: 24 %
% SYSTEM STANDBY
% If the state of this machine is ADS MANUAL and the system is in the SYSTEM STANDBY state, then go to the ADS STANDBY state %
SOR EQU N18:0 N9:43 EQU N10:0 N9:0 MOV N9:40 N18:0 EOR
%   N18:0  ADS_C_STATE  "<datalog>" %
%   N9:43  ADS_MANUAL  "STATE ADS Manual" %
%   N10:0  SYSTEM_STATE  "<datalog> STATE The current state of the system" %
%   N9:0  SYSTEM_STANDBY  "STATE System Standby" %
%   N9:40  ADS_STANDBY  "STATE ADS Standby" %
% Rung: 25 %
% TITLE: ADS ALARM %
% Exiting ADS ALARM
% If the state of this machine is ADS ALARM and the alrms are not active and the buffered state is not ADS STANDBY, then go to the buffered state and clear the buffer %
SOR EQU N18:0 N9:44 EQU N18:5 0 NEQ N18:4 0 BST MOV N18:4 N16:0 NXB MOV 0 N18:4 BND EOR
%   N18:0  ADS_C_STATE  "<datalog>" %
%   N9:44  ADS_ALARM  "STATE ADS Alarm" %
%   N18:5  ADS_C_ALARMS_0 %
%   N18:4  ADS_C_ADS_ALARM_BUFR %
%   N16:0  ADS_A_STATE  "<datalog> STATE The current state of Adsorber A" %
% Rung: 26 %
% Exiting ADS ALARM
% If the state of this machine is ADS ALARM and the alarms are not active and the buffered state is empty, then go to the ADS STANDBY state %
SOR EQU N18:0 N9:44 EQU N18:5 0 EQU N18:4 0 MOV N9:40 N18:0 EOR
%   N18:0  ADS_C_STATE  "<datalog>" %
%   N9:44  ADS_ALARM  "STATE ADS Alarm" %
%   N18:5  ADS_C_ALARMS_0 %
%   N18:4  ADS_C_ADS_ALARM_BUFR %
%   N9:40  ADS_STANDBY  "STATE ADS Standby" %

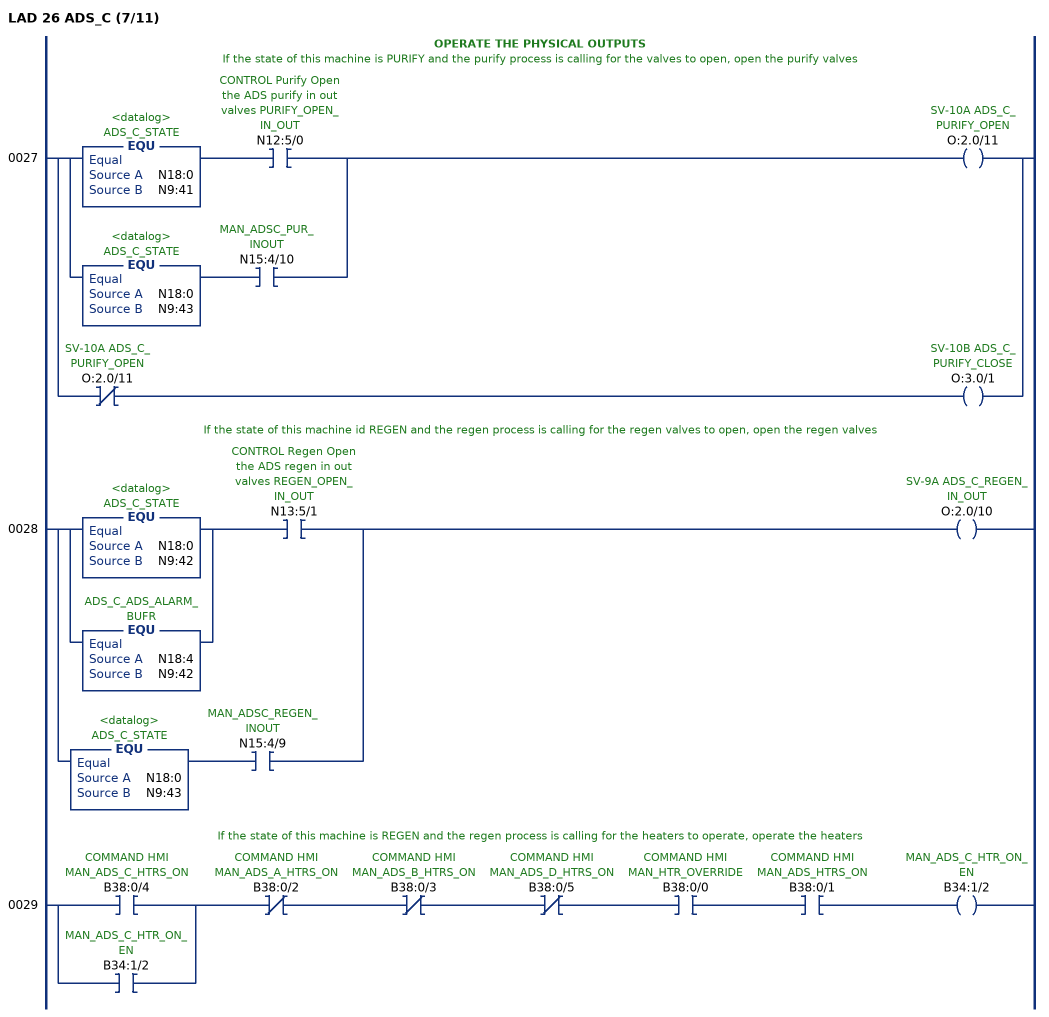
% Rung: 27 %
% TITLE: OPERATE THE PHYSICAL OUTPUTS %
% If the state of this machine is PURIFY and the purify process is calling for the valves to open, open the purify valves %
SOR BST BST EQU N18:0 N9:41 XIC N12:5/0 NXB EQU N18:0 N9:43 XIC N15:4/10 BND OTE O:2.0/11 NXB XIO O:2.0/11 OTE O:3.0/1 BND EOR
%   N18:0  ADS_C_STATE  "<datalog>" %
%   N9:41  ADS_PURIFY  "STATE ADS Purify" %
%   N12:5/0  PURIFY_OPEN_IN_OUT  "CONTROL Purify Open the ADS purify in out valves" %
%   N9:43  ADS_MANUAL  "STATE ADS Manual" %
%   N15:4/10  MAN_ADSC_PUR_INOUT %
%   O:2.0/11  ADS_C_PURIFY_OPEN  "SV-10A" %
%   O:3.0/1  ADS_C_PURIFY_CLOSE  "SV-10B" %
% Rung: 28 %
% If the state of this machine id REGEN and the regen process is calling for the regen valves to open, open the regen valves %
SOR BST BST EQU N18:0 N9:42 NXB EQU N18:4 N9:42 BND XIC N13:5/1 NXB EQU N18:0 N9:43 XIC N15:4/9 BND OTE O:2.0/10 EOR
%   N18:0  ADS_C_STATE  "<datalog>" %
%   N9:42  ADS_REGEN  "STATE ADS Regen" %
%   N18:4  ADS_C_ADS_ALARM_BUFR %
%   N13:5/1  REGEN_OPEN_IN_OUT  "CONTROL Regen Open the ADS regen in out valves" %
%   N9:43  ADS_MANUAL  "STATE ADS Manual" %
%   N15:4/9  MAN_ADSC_REGEN_INOUT %
%   O:2.0/10  ADS_C_REGEN_IN_OUT  "SV-9A" %
% Rung: 29 %
% If the state of this machine is REGEN and the regen process is calling for the heaters to operate, operate the heaters %
SOR BST XIC B38:0/4 NXB XIC B34:1/2 BND XIO B38:0/2 XIO B38:0/3 XIO B38:0/5 XIC B38:0/0 XIC B38:0/1 OTE B34:1/2 EOR
%   B38:0/4  MAN_ADS_C_HTRS_ON  "COMMAND HMI" %
%   B34:1/2  MAN_ADS_C_HTR_ON_EN %
%   B38:0/2  MAN_ADS_A_HTRS_ON  "COMMAND HMI" %
%   B38:0/3  MAN_ADS_B_HTRS_ON  "COMMAND HMI" %
%   B38:0/5  MAN_ADS_D_HTRS_ON  "COMMAND HMI" %
%   B38:0/0  MAN_HTR_OVERRIDE  "COMMAND HMI" %
%   B38:0/1  MAN_ADS_HTRS_ON  "COMMAND HMI" %

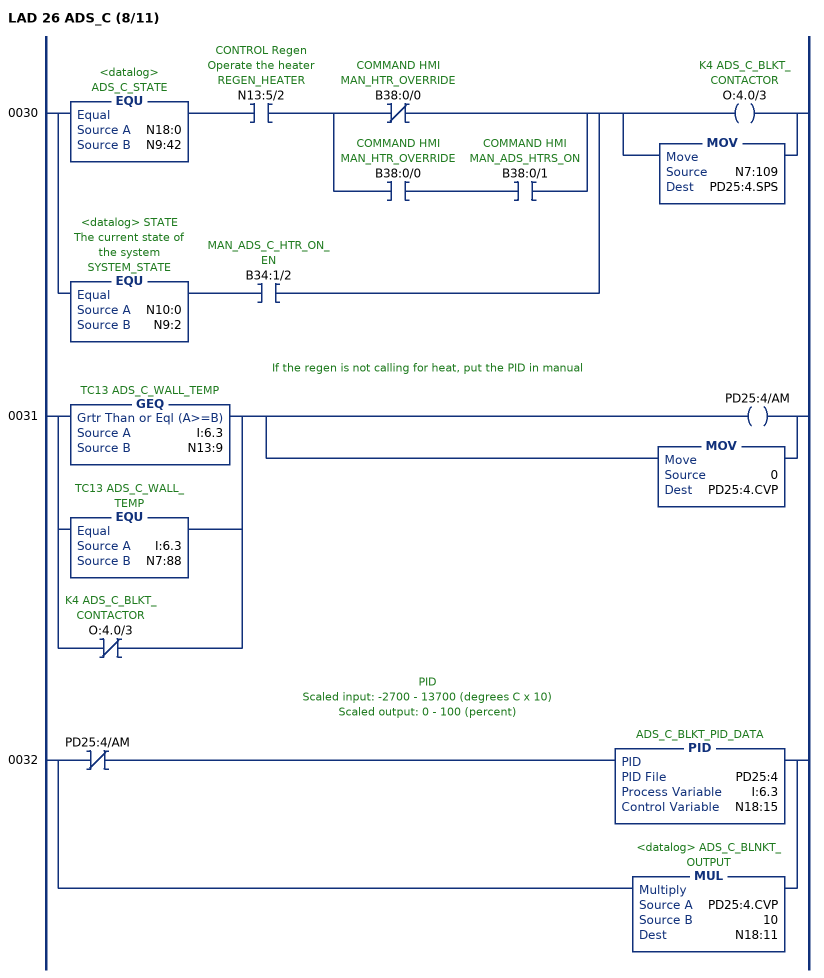
% Rung: 30 %
SOR BST EQU N18:0 N9:42 XIC N13:5/2 BST XIO B38:0/0 NXB XIC B38:0/0 XIC B38:0/1 BND NXB EQU N10:0 N9:2 XIC B34:1/2 BND BST OTE O:4.0/3 NXB MOV N7:109 PD25:4.SPS BND EOR
%   N18:0  ADS_C_STATE  "<datalog>" %
%   N9:42  ADS_REGEN  "STATE ADS Regen" %
%   N13:5/2  REGEN_HEATER  "CONTROL Regen Operate the heater" %
%   B38:0/0  MAN_HTR_OVERRIDE  "COMMAND HMI" %
%   B38:0/1  MAN_ADS_HTRS_ON  "COMMAND HMI" %
%   N10:0  SYSTEM_STATE  "<datalog> STATE The current state of the system" %
%   N9:2  SYSTEM_MANUAL  "STATE System Manual" %
%   B34:1/2  MAN_ADS_C_HTR_ON_EN %
%   O:4.0/3  ADS_C_BLKT_CONTACTOR  "K4" %
%   N7:109  BLANKET_SP  "<datalog> ADS Blanket PID Setpoint" %
% Rung: 31 %
% If the regen is not calling for heat, put the PID in manual %
SOR BST GEQ I:6.3 N13:9 NXB EQU I:6.3 N7:88 NXB XIO O:4.0/3 BND BST OTE PD25:4/AM NXB MOV 0 PD25:4.CVP BND EOR
%   I:6.3  ADS_C_WALL_TEMP  "TC13" %
%   N13:9  BLANKET_LIMIT  "ADS Blanket Temp Limit" %
%   N7:88  TC_OPEN_SP  "CONFIG TC Open Setpoint" %
%   O:4.0/3  ADS_C_BLKT_CONTACTOR  "K4" %
% Rung: 32 %
% PID
% Scaled input: -2700 - 13700 (degrees C x 10)
% Scaled output: 0 - 100 (percent) %
SOR BST XIO PD25:4/AM PID PD25:4 I:6.3 N18:15 NXB MUL PD25:4.CVP 10 N18:11 BND EOR
%   PD25:4  ADS_C_BLKT_PID_DATA %
%   I:6.3  ADS_C_WALL_TEMP  "TC13" %
%   N18:15  ADS_C_BLKT_OUTPT_RAW %
%   N18:11  ADS_C_BLNKT_OUTPUT  "<datalog>" %

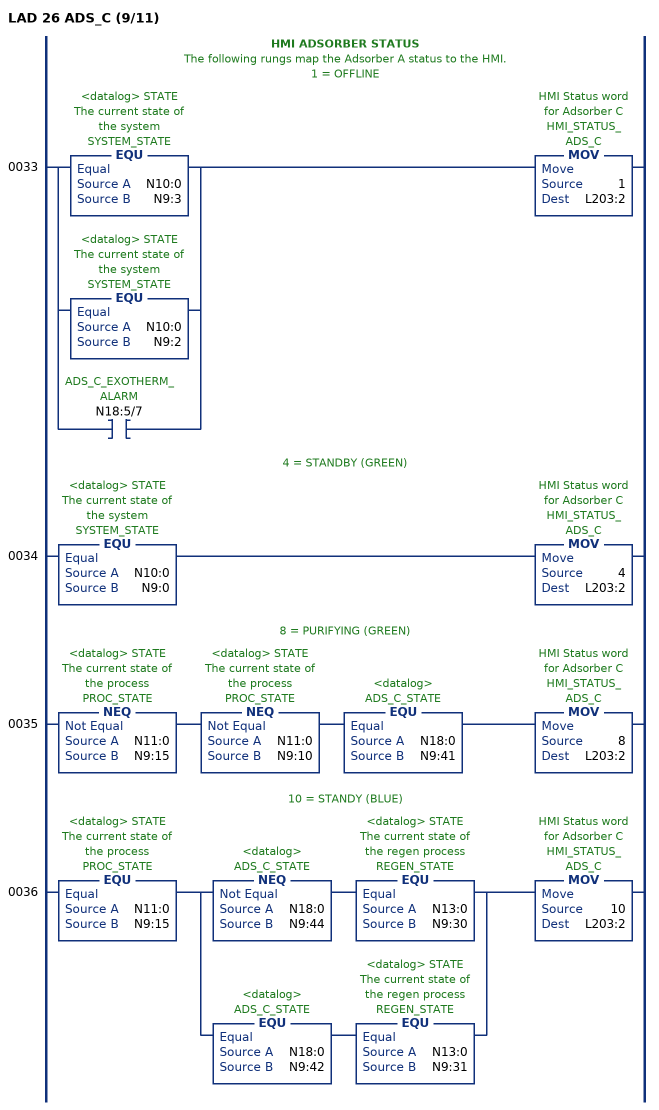
% Rung: 33 %
% TITLE: HMI ADSORBER STATUS %
% The following rungs map the Adsorber A status to the HMI.
% 1 = OFFLINE %
SOR BST EQU N10:0 N9:3 NXB EQU N10:0 N9:2 NXB XIC N18:5/7 BND MOV 1 L203:2 EOR
%   N10:0  SYSTEM_STATE  "<datalog> STATE The current state of the system" %
%   N9:3  SYSTEM_ALARM  "STATE System Alarm" %
%   N9:2  SYSTEM_MANUAL  "STATE System Manual" %
%   N18:5/7  ADS_C_EXOTHERM_ALARM %
%   L203:2  HMI_STATUS_ADS_C  "HMI Status word for Adsorber C" %
% Rung: 34 %
% 4 = STANDBY (GREEN) %
SOR EQU N10:0 N9:0 MOV 4 L203:2 EOR
%   N10:0  SYSTEM_STATE  "<datalog> STATE The current state of the system" %
%   N9:0  SYSTEM_STANDBY  "STATE System Standby" %
%   L203:2  HMI_STATUS_ADS_C  "HMI Status word for Adsorber C" %
% Rung: 35 %
% 8 = PURIFYING (GREEN) %
SOR NEQ N11:0 N9:15 NEQ N11:0 N9:10 EQU N18:0 N9:41 MOV 8 L203:2 EOR
%   N11:0  PROC_STATE  "<datalog> STATE The current state of the process" %
%   N9:15  PROC_REGEN_C  "STATE Process Regen C" %
%   N9:10  PROCESS_STANDBY  "STATE Process Standby" %
%   N18:0  ADS_C_STATE  "<datalog>" %
%   N9:41  ADS_PURIFY  "STATE ADS Purify" %
%   L203:2  HMI_STATUS_ADS_C  "HMI Status word for Adsorber C" %
% Rung: 36 %
% 10 = STANDY (BLUE) %
SOR EQU N11:0 N9:15 BST NEQ N18:0 N9:44 EQU N13:0 N9:30 NXB EQU N18:0 N9:42 EQU N13:0 N9:31 BND MOV 10 L203:2 EOR
%   N11:0  PROC_STATE  "<datalog> STATE The current state of the process" %
%   N9:15  PROC_REGEN_C  "STATE Process Regen C" %
%   N18:0  ADS_C_STATE  "<datalog>" %
%   N9:44  ADS_ALARM  "STATE ADS Alarm" %
%   N13:0  REGEN_STATE  "<datalog> STATE The current state of the regen process" %
%   N9:30  REGEN_STANDBY  "STATE Regen Standby" %
%   N9:42  ADS_REGEN  "STATE ADS Regen" %
%   N9:31  REGEN_DELAY  "STATE Regen Delay" %
%   L203:2  HMI_STATUS_ADS_C  "HMI Status word for Adsorber C" %

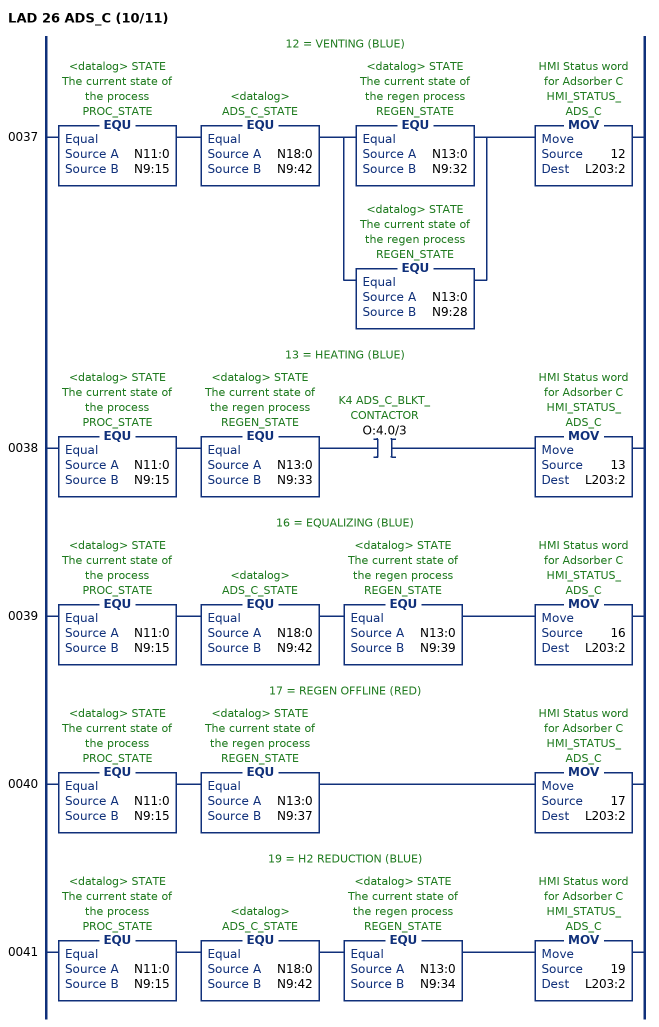
% Rung: 37 %
% 12 = VENTING (BLUE) %
SOR EQU N11:0 N9:15 EQU N18:0 N9:42 BST EQU N13:0 N9:32 NXB EQU N13:0 N9:28 BND MOV 12 L203:2 EOR
%   N11:0  PROC_STATE  "<datalog> STATE The current state of the process" %
%   N9:15  PROC_REGEN_C  "STATE Process Regen C" %
%   N18:0  ADS_C_STATE  "<datalog>" %
%   N9:42  ADS_REGEN  "STATE ADS Regen" %
%   N13:0  REGEN_STATE  "<datalog> STATE The current state of the regen process" %
%   N9:32  REGEN_VENT  "STATE Regen Vent" %
%   N9:28  REGEN_VENT_2 %
%   L203:2  HMI_STATUS_ADS_C  "HMI Status word for Adsorber C" %
% Rung: 38 %
% 13 = HEATING (BLUE) %
SOR EQU N11:0 N9:15 EQU N13:0 N9:33 XIC O:4.0/3 MOV 13 L203:2 EOR
%   N11:0  PROC_STATE  "<datalog> STATE The current state of the process" %
%   N9:15  PROC_REGEN_C  "STATE Process Regen C" %
%   N13:0  REGEN_STATE  "<datalog> STATE The current state of the regen process" %
%   N9:33  REGEN_HEAT_BED  "STATE Regen Heat wall" %
%   O:4.0/3  ADS_C_BLKT_CONTACTOR  "K4" %
%   L203:2  HMI_STATUS_ADS_C  "HMI Status word for Adsorber C" %
% Rung: 39 %
% 16 = EQUALIZING (BLUE) %
SOR EQU N11:0 N9:15 EQU N18:0 N9:42 EQU N13:0 N9:39 MOV 16 L203:2 EOR
%   N11:0  PROC_STATE  "<datalog> STATE The current state of the process" %
%   N9:15  PROC_REGEN_C  "STATE Process Regen C" %
%   N18:0  ADS_C_STATE  "<datalog>" %
%   N9:42  ADS_REGEN  "STATE ADS Regen" %
%   N13:0  REGEN_STATE  "<datalog> STATE The current state of the regen process" %
%   N9:39  REGEN_EQUALIZE  "STATE Regen Equalize" %
%   L203:2  HMI_STATUS_ADS_C  "HMI Status word for Adsorber C" %
% Rung: 40 %
% 17 = REGEN OFFLINE (RED) %
SOR EQU N11:0 N9:15 EQU N13:0 N9:37 MOV 17 L203:2 EOR
%   N11:0  PROC_STATE  "<datalog> STATE The current state of the process" %
%   N9:15  PROC_REGEN_C  "STATE Process Regen C" %
%   N13:0  REGEN_STATE  "<datalog> STATE The current state of the regen process" %
%   N9:37  REGEN_ALARM  "STATE Regen Alarm" %
%   L203:2  HMI_STATUS_ADS_C  "HMI Status word for Adsorber C" %
% Rung: 41 %
% 19 = H2 REDUCTION (BLUE) %
SOR EQU N11:0 N9:15 EQU N18:0 N9:42 EQU N13:0 N9:34 MOV 19 L203:2 EOR
%   N11:0  PROC_STATE  "<datalog> STATE The current state of the process" %
%   N9:15  PROC_REGEN_C  "STATE Process Regen C" %
%   N18:0  ADS_C_STATE  "<datalog>" %
%   N9:42  ADS_REGEN  "STATE ADS Regen" %
%   N13:0  REGEN_STATE  "<datalog> STATE The current state of the regen process" %
%   N9:34  REGEN_H2_REDUCTION  "STATE Regen Running" %
%   L203:2  HMI_STATUS_ADS_C  "HMI Status word for Adsorber C" %

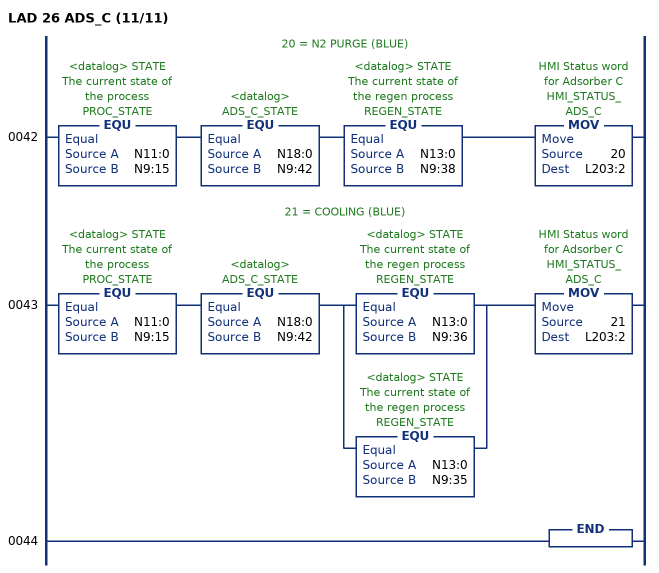
% Rung: 42 %
% 20 = N2 PURGE (BLUE) %
SOR EQU N11:0 N9:15 EQU N18:0 N9:42 EQU N13:0 N9:38 MOV 20 L203:2 EOR
%   N11:0  PROC_STATE  "<datalog> STATE The current state of the process" %
%   N9:15  PROC_REGEN_C  "STATE Process Regen C" %
%   N18:0  ADS_C_STATE  "<datalog>" %
%   N9:42  ADS_REGEN  "STATE ADS Regen" %
%   N13:0  REGEN_STATE  "<datalog> STATE The current state of the regen process" %
%   N9:38  REGEN_PURGE  "STATE Regen Hot Purge" %
%   L203:2  HMI_STATUS_ADS_C  "HMI Status word for Adsorber C" %
% Rung: 43 %
% 21 = COOLING (BLUE) %
SOR EQU N11:0 N9:15 EQU N18:0 N9:42 BST EQU N13:0 N9:36 NXB EQU N13:0 N9:35 BND MOV 21 L203:2 EOR
%   N11:0  PROC_STATE  "<datalog> STATE The current state of the process" %
%   N9:15  PROC_REGEN_C  "STATE Process Regen C" %
%   N18:0  ADS_C_STATE  "<datalog>" %
%   N9:42  ADS_REGEN  "STATE ADS Regen" %
%   N13:0  REGEN_STATE  "<datalog> STATE The current state of the regen process" %
%   N9:36  REGEN_COOL  "STATE Regen Cool" %
%   N9:35  REGEN_COOL_WALL  "STATE Regen Cool wall" %
%   L203:2  HMI_STATUS_ADS_C  "HMI Status word for Adsorber C" %
% Rung: 44 %
SOR END EOR

LADDER 27 "ADS_C_FLT"
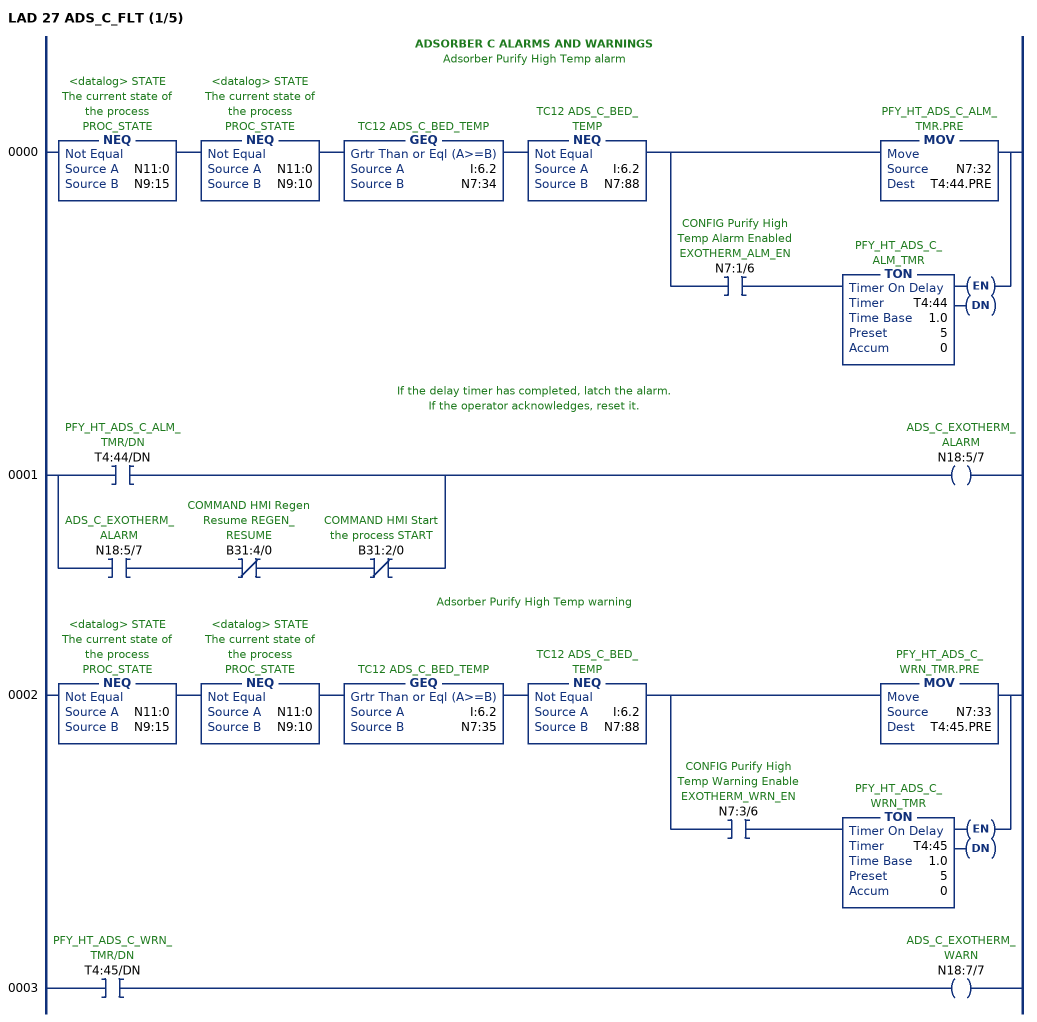
% Rung: 0 %
% TITLE: ADSORBER C ALARMS AND WARNINGS %
% Adsorber Purify High Temp alarm %
SOR NEQ N11:0 N9:15 NEQ N11:0 N9:10 GEQ I:6.2 N7:34 NEQ I:6.2 N7:88 BST MOV N7:32 T4:44.PRE NXB XIC N7:1/6 TON T4:44 1.0 5 0 BND EOR
%   N11:0  PROC_STATE  "<datalog> STATE The current state of the process" %
%   N9:15  PROC_REGEN_C  "STATE Process Regen C" %
%   N9:10  PROCESS_STANDBY  "STATE Process Standby" %
%   I:6.2  ADS_C_BED_TEMP  "TC12" %
%   N7:34  EXOTHERM_ALM_SP  "CONFIG Purify High Temp Alarm Setpoint" %
%   N7:88  TC_OPEN_SP  "CONFIG TC Open Setpoint" %
%   N7:32  EXOTHERM_ALM_DLY  "CONFIG Purify High Temp Alarm Delay" %
%   T4:44  PFY_HT_ADS_C_ALM_TMR %
%   N7:1/6  EXOTHERM_ALM_EN  "CONFIG Purify High Temp Alarm Enabled" %
% Rung: 1 %
% If the delay timer has completed, latch the alarm.
% If the operator acknowledges, reset it. %
SOR BST XIC T4:44/DN NXB XIC N18:5/7 XIO B31:4/0 XIO B31:2/0 BND OTE N18:5/7 EOR
%   T4:44  PFY_HT_ADS_C_ALM_TMR %
%   N18:5/7  ADS_C_EXOTHERM_ALARM %
%   B31:4/0  REGEN_RESUME  "COMMAND HMI Regen Resume" %
%   B31:2/0  START  "COMMAND HMI Start the process" %
% Rung: 2 %
% Adsorber Purify High Temp warning %
SOR NEQ N11:0 N9:15 NEQ N11:0 N9:10 GEQ I:6.2 N7:35 NEQ I:6.2 N7:88 BST MOV N7:33 T4:45.PRE NXB XIC N7:3/6 TON T4:45 1.0 5 0 BND EOR
%   N11:0  PROC_STATE  "<datalog> STATE The current state of the process" %
%   N9:15  PROC_REGEN_C  "STATE Process Regen C" %
%   N9:10  PROCESS_STANDBY  "STATE Process Standby" %
%   I:6.2  ADS_C_BED_TEMP  "TC12" %
%   N7:35  EXOTHERM_WRN_SP  "CONFIG Purify High Temp Warning Setpoint" %
%   N7:88  TC_OPEN_SP  "CONFIG TC Open Setpoint" %
%   N7:33  EXOTHERM_WRN_DLY  "CONFIG Purify High Temp Warning Delay" %
%   T4:45  PFY_HT_ADS_C_WRN_TMR %
%   N7:3/6  EXOTHERM_WRN_EN  "CONFIG Purify High Temp Warning Enable" %
% Rung: 3 %
SOR XIC T4:45/DN OTE N18:7/7 EOR
%   T4:45  PFY_HT_ADS_C_WRN_TMR %
%   N18:7/7  ADS_C_EXOTHERM_WARN %

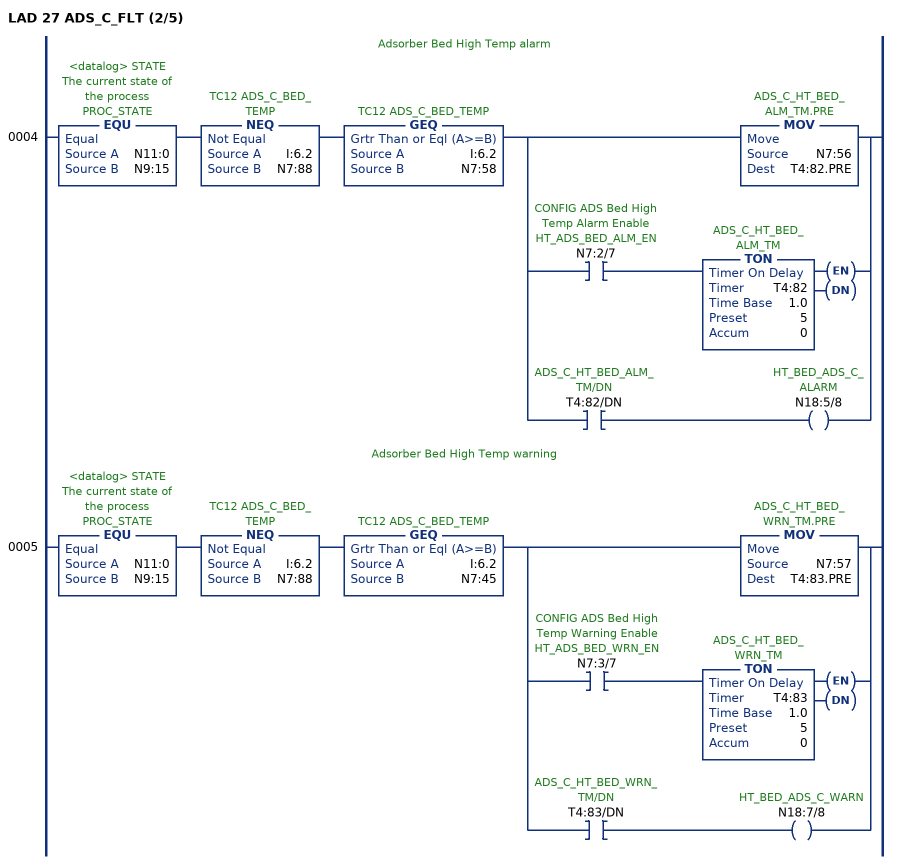
% Rung: 4 %
% Adsorber Bed High Temp alarm %
SOR EQU N11:0 N9:15 NEQ I:6.2 N7:88 GEQ I:6.2 N7:58 BST MOV N7:56 T4:82.PRE NXB XIC N7:2/7 TON T4:82 1.0 5 0 NXB XIC T4:82/DN OTE N18:5/8 BND EOR
%   N11:0  PROC_STATE  "<datalog> STATE The current state of the process" %
%   N9:15  PROC_REGEN_C  "STATE Process Regen C" %
%   I:6.2  ADS_C_BED_TEMP  "TC12" %
%   N7:88  TC_OPEN_SP  "CONFIG TC Open Setpoint" %
%   N7:58  HT_ADS_BED_ALM_SP  "CONFIG ADS Bed High Temp Alarm Setpoint" %
%   N7:56  HT_ADS_BED_ALM_DLY  "CONFIG ADS Bed High Temp Alarm Delay" %
%   T4:82  ADS_C_HT_BED_ALM_TM %
%   N7:2/7  HT_ADS_BED_ALM_EN  "CONFIG ADS Bed High Temp Alarm Enable" %
%   N18:5/8  HT_BED_ADS_C_ALARM %
% Rung: 5 %
% Adsorber Bed High Temp warning %
SOR EQU N11:0 N9:15 NEQ I:6.2 N7:88 GEQ I:6.2 N7:45 BST MOV N7:57 T4:83.PRE NXB XIC N7:3/7 TON T4:83 1.0 5 0 NXB XIC T4:83/DN OTE N18:7/8 BND EOR
%   N11:0  PROC_STATE  "<datalog> STATE The current state of the process" %
%   N9:15  PROC_REGEN_C  "STATE Process Regen C" %
%   I:6.2  ADS_C_BED_TEMP  "TC12" %
%   N7:88  TC_OPEN_SP  "CONFIG TC Open Setpoint" %
%   N7:45  LT_ADS_BED_WRN_SP  "CONFIG ADS Bed Low Temp Warning Setpoint" %
%   N7:57  HT_ADS_BED_WRN_DLY  "CONFIG ADS Bed High Temp Warning Delay" %
%   T4:83  ADS_C_HT_BED_WRN_TM %
%   N7:3/7  HT_ADS_BED_WRN_EN  "CONFIG ADS Bed High Temp Warning Enable" %
%   N18:7/8  HT_BED_ADS_C_WARN %

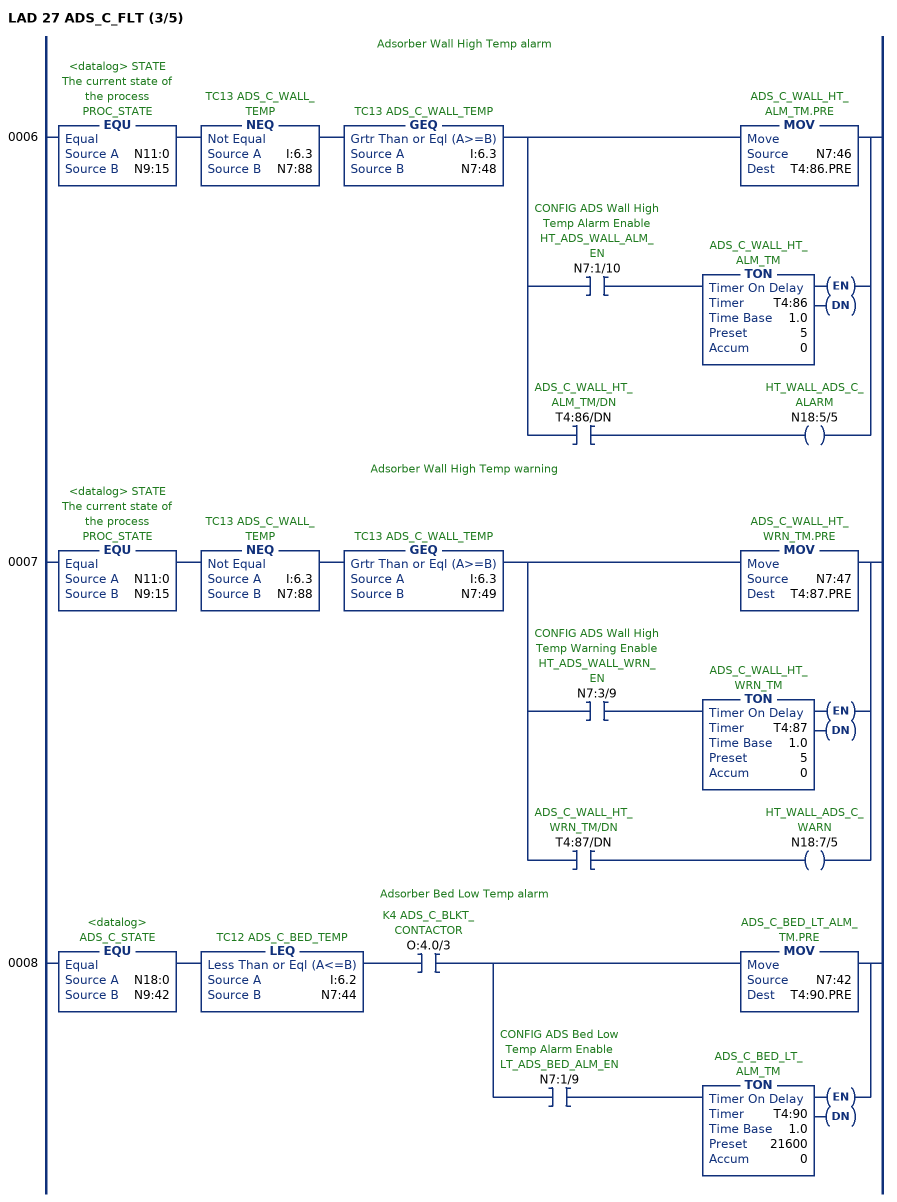
% Rung: 6 %
% Adsorber Wall High Temp alarm %
SOR EQU N11:0 N9:15 NEQ I:6.3 N7:88 GEQ I:6.3 N7:48 BST MOV N7:46 T4:86.PRE NXB XIC N7:1/10 TON T4:86 1.0 5 0 NXB XIC T4:86/DN OTE N18:5/5 BND EOR
%   N11:0  PROC_STATE  "<datalog> STATE The current state of the process" %
%   N9:15  PROC_REGEN_C  "STATE Process Regen C" %
%   I:6.3  ADS_C_WALL_TEMP  "TC13" %
%   N7:88  TC_OPEN_SP  "CONFIG TC Open Setpoint" %
%   N7:48  HT_ADS_WALL_ALM_SP  "CONFIG ADS Wall High Temp Alarm Setpoint" %
%   N7:46  HT_ADS_WALL_ALM_DLY  "CONFIG ADS Wall High Temp Alarm Delay" %
%   T4:86  ADS_C_WALL_HT_ALM_TM %
%   N7:1/10  HT_ADS_WALL_ALM_EN  "CONFIG ADS Wall High Temp Alarm Enable" %
%   N18:5/5  HT_WALL_ADS_C_ALARM %
% Rung: 7 %
% Adsorber Wall High Temp warning %
SOR EQU N11:0 N9:15 NEQ I:6.3 N7:88 GEQ I:6.3 N7:49 BST MOV N7:47 T4:87.PRE NXB XIC N7:3/9 TON T4:87 1.0 5 0 NXB XIC T4:87/DN OTE N18:7/5 BND EOR
%   N11:0  PROC_STATE  "<datalog> STATE The current state of the process" %
%   N9:15  PROC_REGEN_C  "STATE Process Regen C" %
%   I:6.3  ADS_C_WALL_TEMP  "TC13" %
%   N7:88  TC_OPEN_SP  "CONFIG TC Open Setpoint" %
%   N7:49  HT_ADS_WALL_WRN_SP  "CONFIG ADS Wall High Temp Warning Setpoint" %
%   N7:47  HT_ADS_WALL_WRN_DLY  "CONFIG ADS Wall High Temp Warning Delay" %
%   T4:87  ADS_C_WALL_HT_WRN_TM %
%   N7:3/9  HT_ADS_WALL_WRN_EN  "CONFIG ADS Wall High Temp Warning Enable" %
%   N18:7/5  HT_WALL_ADS_C_WARN %
% Rung: 8 %
% Adsorber Bed Low Temp alarm %
SOR EQU N18:0 N9:42 LEQ I:6.2 N7:44 XIC O:4.0/3 BST MOV N7:42 T4:90.PRE NXB XIC N7:1/9 TON T4:90 1.0 21600 0 BND EOR
%   N18:0  ADS_C_STATE  "<datalog>" %
%   N9:42  ADS_REGEN  "STATE ADS Regen" %
%   I:6.2  ADS_C_BED_TEMP  "TC12" %
%   N7:44  LT_ADS_BED_ALM_SP  "CONFIG ADS Bed Low Temp Alarm Setpoint" %
%   O:4.0/3  ADS_C_BLKT_CONTACTOR  "K4" %
%   N7:42  LT_ADS_BED_ALM_DLY  "CONFIG ADS Bed Low Temp Alarm Delay" %
%   T4:90  ADS_C_BED_LT_ALM_TM %
%   N7:1/9  LT_ADS_BED_ALM_EN  "CONFIG ADS Bed Low Temp Alarm Enable" %

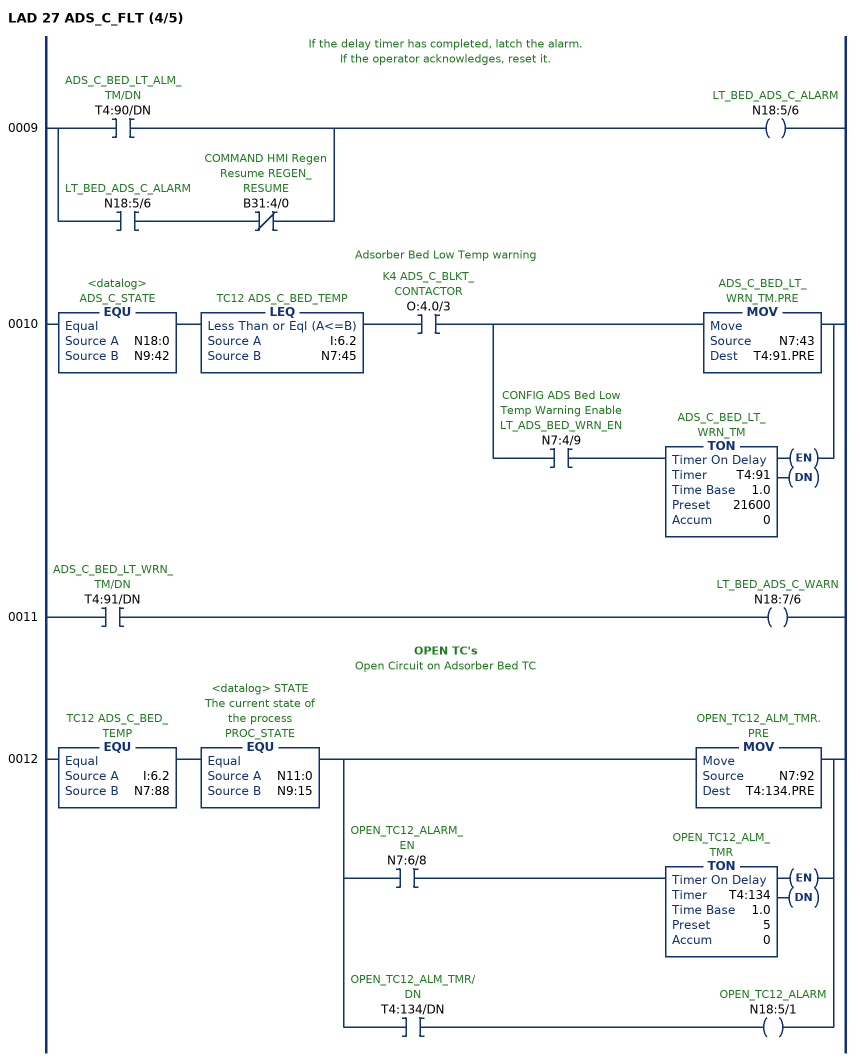
% Rung: 9 %
% If the delay timer has completed, latch the alarm.
% If the operator acknowledges, reset it. %
SOR BST XIC T4:90/DN NXB XIC N18:5/6 XIO B31:4/0 BND OTE N18:5/6 EOR
%   T4:90  ADS_C_BED_LT_ALM_TM %
%   N18:5/6  LT_BED_ADS_C_ALARM %
%   B31:4/0  REGEN_RESUME  "COMMAND HMI Regen Resume" %
% Rung: 10 %
% Adsorber Bed Low Temp warning %
SOR EQU N18:0 N9:42 LEQ I:6.2 N7:45 XIC O:4.0/3 BST MOV N7:43 T4:91.PRE NXB XIC N7:4/9 TON T4:91 1.0 21600 0 BND EOR
%   N18:0  ADS_C_STATE  "<datalog>" %
%   N9:42  ADS_REGEN  "STATE ADS Regen" %
%   I:6.2  ADS_C_BED_TEMP  "TC12" %
%   N7:45  LT_ADS_BED_WRN_SP  "CONFIG ADS Bed Low Temp Warning Setpoint" %
%   O:4.0/3  ADS_C_BLKT_CONTACTOR  "K4" %
%   N7:43  LT_ADS_BED_WRN_DLY  "CONFIG ADS Bed Low Temp Warning Delay" %
%   T4:91  ADS_C_BED_LT_WRN_TM %
%   N7:4/9  LT_ADS_BED_WRN_EN  "CONFIG ADS Bed Low Temp Warning Enable" %
% Rung: 11 %
SOR XIC T4:91/DN OTE N18:7/6 EOR
%   T4:91  ADS_C_BED_LT_WRN_TM %
%   N18:7/6  LT_BED_ADS_C_WARN %
% Rung: 12 %
% TITLE: OPEN TC's %
% Open Circuit on Adsorber Bed TC %
SOR EQU I:6.2 N7:88 EQU N11:0 N9:15 BST MOV N7:92 T4:134.PRE NXB XIC N7:6/8 TON T4:134 1.0 5 0 NXB XIC T4:134/DN OTE N18:5/1 BND EOR
%   I:6.2  ADS_C_BED_TEMP  "TC12" %
%   N7:88  TC_OPEN_SP  "CONFIG TC Open Setpoint" %
%   N11:0  PROC_STATE  "<datalog> STATE The current state of the process" %
%   N9:15  PROC_REGEN_C  "STATE Process Regen C" %
%   N7:92  OPEN_TC_ALM_DLY  "CONFIG TC Open Alarm Delay" %
%   T4:134  OPEN_TC12_ALM_TMR %
%   N7:6/8  OPEN_TC12_ALARM_EN %
%   N18:5/1  OPEN_TC12_ALARM %

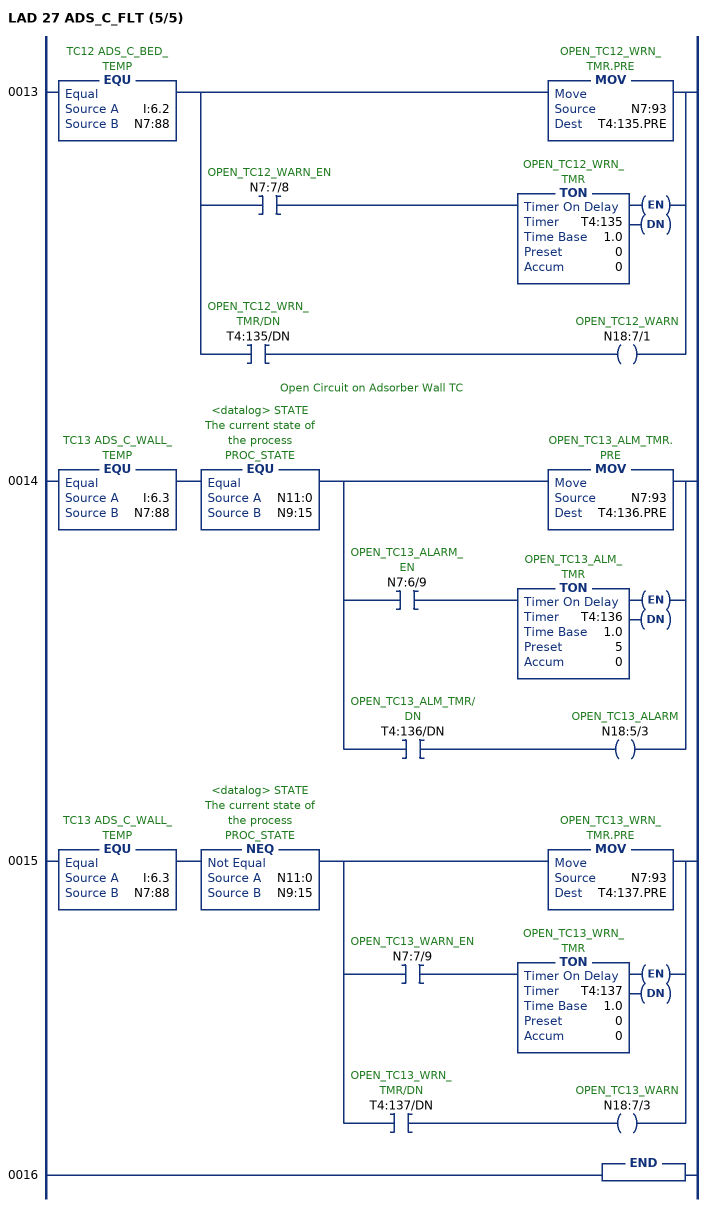
% Rung: 13 %
SOR EQU I:6.2 N7:88 BST MOV N7:93 T4:135.PRE NXB XIC N7:7/8 TON T4:135 1.0 0 0 NXB XIC T4:135/DN OTE N18:7/1 BND EOR
%   I:6.2  ADS_C_BED_TEMP  "TC12" %
%   N7:88  TC_OPEN_SP  "CONFIG TC Open Setpoint" %
%   N7:93  OPEN_TC_WRN_DLY  "CONFIG TC Open Warning Delay" %
%   T4:135  OPEN_TC12_WRN_TMR %
%   N7:7/8  OPEN_TC12_WARN_EN %
%   N18:7/1  OPEN_TC12_WARN %
% Rung: 14 %
% Open Circuit on Adsorber Wall TC %
SOR EQU I:6.3 N7:88 EQU N11:0 N9:15 BST MOV N7:93 T4:136.PRE NXB XIC N7:6/9 TON T4:136 1.0 5 0 NXB XIC T4:136/DN OTE N18:5/3 BND EOR
%   I:6.3  ADS_C_WALL_TEMP  "TC13" %
%   N7:88  TC_OPEN_SP  "CONFIG TC Open Setpoint" %
%   N11:0  PROC_STATE  "<datalog> STATE The current state of the process" %
%   N9:15  PROC_REGEN_C  "STATE Process Regen C" %
%   N7:93  OPEN_TC_WRN_DLY  "CONFIG TC Open Warning Delay" %
%   T4:136  OPEN_TC13_ALM_TMR %
%   N7:6/9  OPEN_TC13_ALARM_EN %
%   N18:5/3  OPEN_TC13_ALARM %
% Rung: 15 %
SOR EQU I:6.3 N7:88 NEQ N11:0 N9:15 BST MOV N7:93 T4:137.PRE NXB XIC N7:7/9 TON T4:137 1.0 0 0 NXB XIC T4:137/DN OTE N18:7/3 BND EOR
%   I:6.3  ADS_C_WALL_TEMP  "TC13" %
%   N7:88  TC_OPEN_SP  "CONFIG TC Open Setpoint" %
%   N11:0  PROC_STATE  "<datalog> STATE The current state of the process" %
%   N9:15  PROC_REGEN_C  "STATE Process Regen C" %
%   N7:93  OPEN_TC_WRN_DLY  "CONFIG TC Open Warning Delay" %
%   T4:137  OPEN_TC13_WRN_TMR %
%   N7:7/9  OPEN_TC13_WARN_EN %
%   N18:7/3  OPEN_TC13_WARN %
% Rung: 16 %
SOR END EOR

LADDER 28 "ADS_D"
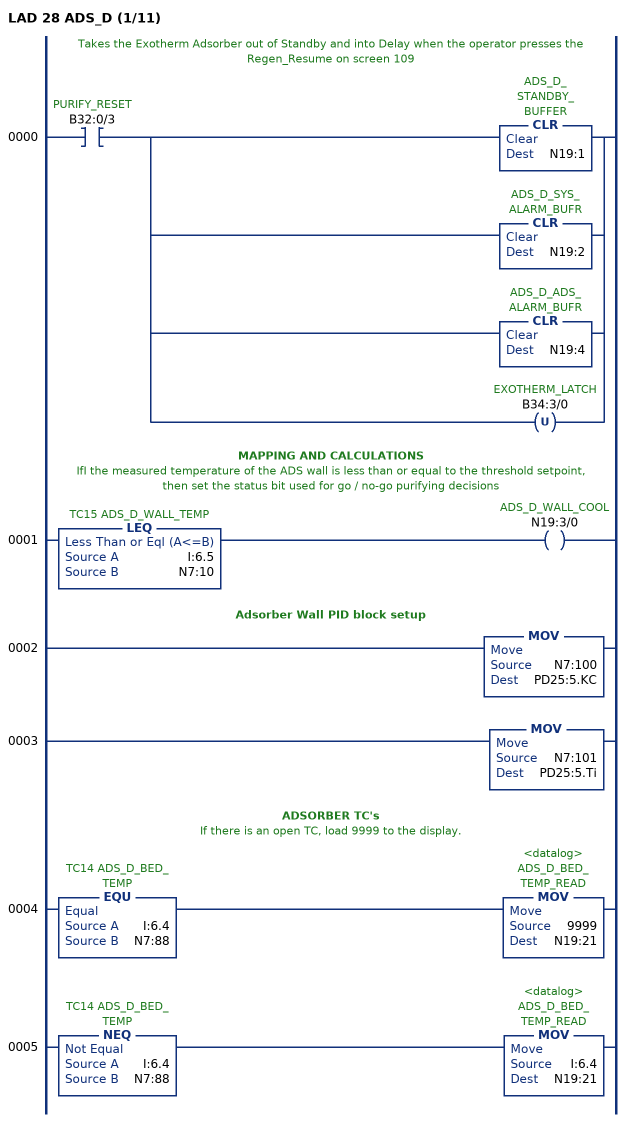
% Rung: 0 %
% Takes the Exotherm Adsorber out of Standby and into Delay when the operator presses the Regen_Resume on screen 109 %
SOR XIC B32:0/3 BST CLR N19:1 NXB CLR N19:2 NXB CLR N19:4 NXB OTU B34:3/0 BND EOR
%   B32:0/3  PURIFY_RESET %
%   N19:1  ADS_D_STANDBY_BUFFER %
%   N19:2  ADS_D_SYS_ALARM_BUFR %
%   N19:4  ADS_D_ADS_ALARM_BUFR %
%   B34:3/0  EXOTHERM_LATCH %
% Rung: 1 %
% TITLE: MAPPING AND CALCULATIONS %
% IfI the measured temperature of the ADS wall is less than or equal to the threshold setpoint, then set the status bit used for go / no-go purifying decisions %
SOR LEQ I:6.5 N7:10 OTE N19:3/0 EOR
%   I:6.5  ADS_D_WALL_TEMP  "TC15" %
%   N7:10  ADS_WALL_TEMP_COOL  "CONFIG The temp at which the adsorber wall is deemed to be cool enough to purify" %
%   N19:3/0  ADS_D_WALL_COOL %
% Rung: 2 %
% TITLE: Adsorber Wall PID block setup %
SOR MOV N7:100 PD25:5.KC EOR
%   N7:100  BLANKET_P  "CONFIG Blanket Proportional Gain" %
% Rung: 3 %
SOR MOV N7:101 PD25:5.Ti EOR
%   N7:101  BLANKET_I  "CONFIG Blanket Integral Gain" %
% Rung: 4 %
% TITLE: ADSORBER TC's %
% If there is an open TC, load 9999 to the display. %
SOR EQU I:6.4 N7:88 MOV 9999 N19:21 EOR
%   I:6.4  ADS_D_BED_TEMP  "TC14" %
%   N7:88  TC_OPEN_SP  "CONFIG TC Open Setpoint" %
%   N19:21  ADS_D_BED_TEMP_READ  "<datalog>" %
% Rung: 5 %
SOR NEQ I:6.4 N7:88 MOV I:6.4 N19:21 EOR
%   I:6.4  ADS_D_BED_TEMP  "TC14" %
%   N7:88  TC_OPEN_SP  "CONFIG TC Open Setpoint" %
%   N19:21  ADS_D_BED_TEMP_READ  "<datalog>" %

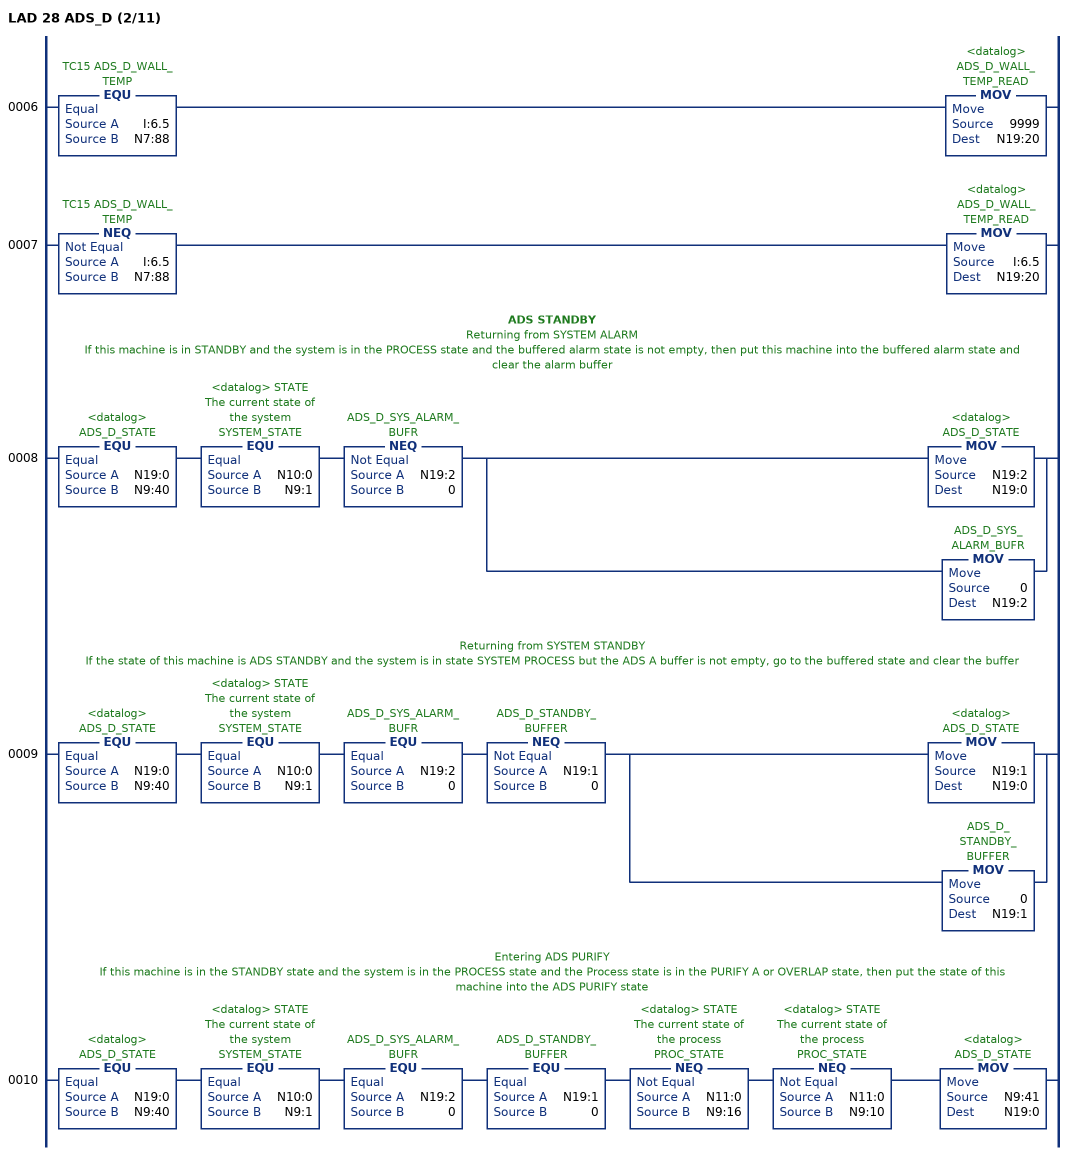
% Rung: 6 %
SOR EQU I:6.5 N7:88 MOV 9999 N19:20 EOR
%   I:6.5  ADS_D_WALL_TEMP  "TC15" %
%   N7:88  TC_OPEN_SP  "CONFIG TC Open Setpoint" %
%   N19:20  ADS_D_WALL_TEMP_READ  "<datalog>" %
% Rung: 7 %
SOR NEQ I:6.5 N7:88 MOV I:6.5 N19:20 EOR
%   I:6.5  ADS_D_WALL_TEMP  "TC15" %
%   N7:88  TC_OPEN_SP  "CONFIG TC Open Setpoint" %
%   N19:20  ADS_D_WALL_TEMP_READ  "<datalog>" %
% Rung: 8 %
% TITLE: ADS STANDBY %
% Returning from SYSTEM ALARM
% If this machine is in STANDBY and the system is in the PROCESS state and the buffered alarm state is not empty, then put this machine into the buffered alarm state and clear the alarm buffer %
SOR EQU N19:0 N9:40 EQU N10:0 N9:1 NEQ N19:2 0 BST MOV N19:2 N19:0 NXB MOV 0 N19:2 BND EOR
%   N19:0  ADS_D_STATE  "<datalog>" %
%   N9:40  ADS_STANDBY  "STATE ADS Standby" %
%   N10:0  SYSTEM_STATE  "<datalog> STATE The current state of the system" %
%   N9:1  SYSTEM_PROCESS  "STATE System Process" %
%   N19:2  ADS_D_SYS_ALARM_BUFR %
% Rung: 9 %
% Returning from SYSTEM STANDBY
% If the state of this machine is ADS STANDBY and the system is in state SYSTEM PROCESS but the ADS A buffer is not empty, go to the buffered state and clear the buffer %
SOR EQU N19:0 N9:40 EQU N10:0 N9:1 EQU N19:2 0 NEQ N19:1 0 BST MOV N19:1 N19:0 NXB MOV 0 N19:1 BND EOR
%   N19:0  ADS_D_STATE  "<datalog>" %
%   N9:40  ADS_STANDBY  "STATE ADS Standby" %
%   N10:0  SYSTEM_STATE  "<datalog> STATE The current state of the system" %
%   N9:1  SYSTEM_PROCESS  "STATE System Process" %
%   N19:2  ADS_D_SYS_ALARM_BUFR %
%   N19:1  ADS_D_STANDBY_BUFFER %
% Rung: 10 %
% Entering ADS PURIFY
% If this machine is in the STANDBY state and the system is in the PROCESS state and the Process state is in the PURIFY A or OVERLAP state, then put the state of this machine into the ADS PURIFY state %
SOR EQU N19:0 N9:40 EQU N10:0 N9:1 EQU N19:2 0 EQU N19:1 0 NEQ N11:0 N9:16 NEQ N11:0 N9:10 MOV N9:41 N19:0 EOR
%   N19:0  ADS_D_STATE  "<datalog>" %
%   N9:40  ADS_STANDBY  "STATE ADS Standby" %
%   N10:0  SYSTEM_STATE  "<datalog> STATE The current state of the system" %
%   N9:1  SYSTEM_PROCESS  "STATE System Process" %
%   N19:2  ADS_D_SYS_ALARM_BUFR %
%   N19:1  ADS_D_STANDBY_BUFFER %
%   N11:0  PROC_STATE  "<datalog> STATE The current state of the process" %
%   N9:16  PROC_REGEN_D  "STATE Process Regen D" %
%   N9:10  PROCESS_STANDBY  "STATE Process Standby" %
%   N9:41  ADS_PURIFY  "STATE ADS Purify" %

